    en_static_define_state_off                      : INT;   // Definierter State für OFF-Zustand
    en_static_define_sub_state_off                  : INT;   // Definierter Substate für OFF-Zustand
    en_static_define_lockdown                       : INT;   // State für Lockdown-Bedingungen
    en_static_define_substate_check_new_state       : INT;   // Substate zur Prüfung eines neuen State
    en_static_define_engine_release_from_substate   : INT;   // Substate, wenn Engine in Release-ON gehen soll
	en_static_define_engine_release_off_substate    : INT;   // Substate, wenn Engine in Release-OFF gehen soll
END_VAR

VAR_OUTPUT
    iAvaiable                                       : INT;   // Verfügbarkeitskennzahl der Engine/Gruppe
    en_available                                    : INT;   // Haupt-State der Verfügbarkeit
    en_available_substate                           : INT;   // Substate der Verfügbarkeit

    iAcknowledge                                    : INT;   // Integer-Wert zur Acknowledge-Verarbeitung
    rAcknowledge                                    : REAL;  // Realwert für Acknowledge-Parameter
    en_acknowledge                                  : INT;   // State für Acknowledge-Vorgang
    en_acknowledge_substate                         : INT;   // Substate des Acknowledge-Vorgangs

    en_demand                                       : INT;   // Haupt-State für Demand-/Anforderung
    en_demand_substate                              : INT;   // Substate für Demand-/Anforderung
    
    ITF_MANAGER                                     : ITF_MANAGER; // Manager-Interface für Gruppen-/Engine-Steuerung
END_VAR

VAR
    aydiSyncG                                       : ARRAY[1..GVL_CONSTANT.MAX_GROUPS] OF DINT := [GVL_CONSTANT.MAX_GROUPS(1)];
                                                        // Array zur Synchronisationsverwaltung der Gruppen

    groups                                          : ARRAY[1..GVL_CONSTANT.MAX_GROUPS] OF ARRAY[0..40] OF ITF_GROUPBASE;
                                                        // Struktur aller Gruppen und ihrer Members

    groups_en_available                             : ARRAY[1..GVL_CONSTANT.MAX_GROUPS] OF INT; // Verfügbarkeits-State je Gruppe
    groups_en_available_old                         : ARRAY[1..GVL_CONSTANT.MAX_GROUPS] OF INT; // Vorheriger Verfügbarkeits-State
    groups_en_available_substate                    : ARRAY[1..GVL_CONSTANT.MAX_GROUPS] OF INT; // Verfügbarkeits-Substate je Gruppe
    groups_en_available_substate_old                : ARRAY[1..GVL_CONSTANT.MAX_GROUPS] OF INT; // Alter Substate

    groups_engine_avaiable                          : ARRAY[1..GVL_CONSTANT.MAX_GROUPS] OF INT; // Engine-Verfügbarkeitsstate je Gruppe

    groups_en_acknowledge                           : ARRAY[1..GVL_CONSTANT.MAX_GROUPS] OF INT; // Acknowledge-State je Gruppe
    groups_en_acknowledge_old                       : ARRAY[1..GVL_CONSTANT.MAX_GROUPS] OF INT; // Alter Acknowledge-State
    groups_en_acknowledge_substate                  : ARRAY[1..GVL_CONSTANT.MAX_GROUPS] OF INT; // Acknowledge-Substate je Gruppe
    groups_en_acknowledge_substate_old              : ARRAY[1..GVL_CONSTANT.MAX_GROUPS] OF INT; // Alter Acknowledge-Substate

    groups_engine_acknowledge                       : ARRAY[1..GVL_CONSTANT.MAX_GROUPS] OF INT; // Engine-Acknowledge-State je Gruppe

    groups_en_release                               : ARRAY[1..GVL_CONSTANT.MAX_GROUPS] OF INT; // Release-State je Gruppe

    AY_GROUPS_AyPosMaxCT                            : ARRAY[1..GVL_CONSTANT.MAX_GROUPS] OF DINT; // Max-CT-Werte der Gruppen
    AY_GROUPS_xReleaseCircuit                       : ARRAY[1..GVL_CONSTANT.MAX_GROUPS] OF BOOL; // Release-Freigabe je Circuit

    TEMP_ITF_GROUPBASE                              : ITF_GROUPBASE; // Temp-Objekt für Gruppenoperationen
    TEMP_ITF_CIRCUIT                                : ITF_CIRCUIT;    // Temp-Circuit-Objekt
    TEMP_ITF_HYDRA                                  : ITF_HYDRA;      // Temp-Hydra-Objekt
    TEMP_ITF_HYDRA_MAX_CT                           : ITF_HYDRA;      // Temp-Hydra Objekt für max CT-Ermittlung

    diTempMemberCount                                : DINT;  // Temporäre Anzahl an Gruppenmitgliedern
    diFor1                                           : DINT;  // Schleifenzähler 1
    diFor2                                           : DINT;  // Schleifenzähler 2
    diFor3                                           : DINT;  // Schleifenzähler 3
    diNextCircuitToRun                               : DINT;  // Nächster Circuit, der gestartet werden soll
    diNextEngineToRun                                : DINT;  // Nächste Engine, die starten soll
    diNextCircuitToOff                               : DINT;  // Nächster Circuit zum Ausschalten
    diNextEngineToOff                                : DINT;  // Nächste Engine zum Ausschalten

    xTrigOn                                          : BOOL;  // Trigger für Start-/ON-Übergang
    xTrigOff                                         : BOOL;  // Trigger für Stop-/OFF-Übergang
    iTrigOffCount                                    : INT;   // Zähler für OFF-Triggerpflege
    iTrigOffMax                                      : INT;   // Maximal zulässige OFF-Triggerzeit

    enCheckOld                                       : INT;   // Alter Check-State
    enReleaseOld                                     : INT;   // Alter Release-State

    uiCountGroupLockDown                             : UINT;  // Anzahl Gruppen im Lockdown
    uiCountEngineLockDown                            : UINT;  // Anzahl Engines im Lockdown
    uiCountEngineAcknowledge                         : UINT;  // Anzahl Engines, die Acknowledge benötigen
    uiCountGroupLockDownOld                          : UINT;  // Vorherige Lockdown-Gruppenzahl
    uiCountEngineAcknowledgeOld                      : UINT;  // Vorherige Anzahl Acknowledge-Engines
    uiCountEngineLockDownOld                         : UINT;  // Vorherige Lockdown-Enginezahl

    iReleaseOld                                      : INT;   // Alter Releasewert
    iAcknowledgeOld                                  : INT;   // Alter Acknowledgewert

    xReleaseStopp                                    : BOOL;  // Stopp-Bedingung für Release
    TP_ReleaseLock                                   : Standard.TP;   // Timerbaustein für Release-Lock
    xResettReleaseLock_VIS                           : BOOL;  // Reset über VIS zum ReleaseLock

    lock_if_released_in_other_circuit                : BOOL;  // Lock, wenn Release in anderem Circuit aktiv ist

    // Parameter
    fbConfigFile                                     : CtaSysConfig.fbConfigFile; // Konfigurationsdatei-Handler
    scParameter                                      : scParameter;               // Parametrierobjekt
END_VAR

actParameter();

(* ITF *)
ITF_MANAGER := THIS^;

(* CHECK *)
CHECK();

(* AVAIABLE *)
AVAIABLE(); 

(* LOCKDOWN *)
LOCKDOWN();

(* ACKNOWLEDGE *)
ACKNOWLEDGE();

(* MANAGEMENT *)
MANAGEMENT();

(* RELEASE *)
RELEASE();

(* CHECK CHANGE *)
CHECK_RELEASE_CHANGE();

(* UPDATE *)
UPDATE_AT_THE_END();

ACTION CHECK:
(* Set Check State *)
FOR diFor1 := LOWER_BOUND(groups,1) TO UPPER_BOUND(groups,1) DO
	FOR diFor2 := LOWER_BOUND(groups[diFor1],1) TO UPPER_BOUND(groups[diFor1],1) DO
		IF __QUERYINTERFACE(groups[diFor1][diFor2],TEMP_ITF_GROUPBASE) THEN
			TEMP_ITF_GROUPBASE.set_check			(en_check);
			TEMP_ITF_GROUPBASE.set_check_substate	(en_check_substate);
		END_IF;
	END_FOR;
END_FOR;
END_ACTION

METHOD GET_NEXT_ENGINE_TO_RUN 
VAR_INPUT
	enTYPE_OF_ENGINE_MANAGEMENT	:	TYPE_OF_ENGINE_MANAGEMENT;
END_VAR
VAR_OUTPUT
	diNextCircuitToRunOut  		: DINT;
	diNextEngineToRunOut		: DINT;	
END_VAR
VAR 
	_diNextCircuitToRun  		: DINT;
	_diEngineLowestRunTime		: DINT;
	_xAvaiable					: BOOL;
	_xRelease					: BOOL;
	_rRelease					: REAL;
	_xAcknowledge				: BOOL;
	_rAcknowledge				: REAL;
	_xLockDown					: BOOL;
	_udiRunTime		    		: UDINT;
	_udiRunTimeTillOn   		: UDINT;
	_udiMinRunTime				: UDINT;
	_uiLowestWorkloadCircuit	: UINT;
END_VAR
(* Set Min Run Time To Max *)
_udiMinRunTime := 16#FFFFFFFF;
(* Set Lowest Workload Circuit to MAX *)
_uiLowestWorkloadCircuit := 16#FFFF;
(* Set Circuit to 0 *)
_diNextCircuitToRun := 0;
diNextCircuitToRunOut := 0;
(* Set Engine to 0  *)
_diEngineLowestRunTime := 0;
diNextEngineToRunOut := 0;

IF enTYPE_OF_ENGINE_MANAGEMENT = TYPE_OF_ENGINE_MANAGEMENT.RUN_1BY1 THEN
	FOR diFor1 := UPPER_BOUND(groups,1) TO LOWER_BOUND(groups,1) BY -1 DO 
		(* If No Error avaiable to release*)
		IF groups_en_available[diFor1] = en_release  OR groups_en_acknowledge[diFor1] = en_release THEN		
			IF __QUERYINTERFACE(groups[diFor1][LOWER_BOUND(groups[diFor1],1)],TEMP_ITF_CIRCUIT) THEN
				IF TEMP_ITF_CIRCUIT.GET_ANZ_RELEASE > 0 AND TEMP_ITF_CIRCUIT.GET_ANZ_AVAIABLE > 0 THEN
					(* iterate Engine and Check if Avaiable and get the Minits *)
					FOR diFor2 := TEMP_ITF_CIRCUIT.UPPERBOUND TO TEMP_ITF_CIRCUIT.LOWERBOUND BY -1 DO
						TEMP_ITF_CIRCUIT.GET_ENGINE_STATE(	usiNr 			:= TO_USINT(diFor2),
															xAvaiable 		=> _xAvaiable,
															xRelease		=> _xRelease,
															rRelease		=> _rRelease,
															xAcknowledge 	=> _xAcknowledge,
															rAcknowledge 	=> _rAcknowledge,
															xLockDown 		=> _xLockDown,
															udiRunTime 		=> _udiRunTime,
															udiRunTimeTillOn=> _udiRunTimeTillOn);
						(* Get time if Avaiable *)
						IF _xAvaiable AND NOT _xRelease AND NOT _xLockDown THEN
							IF _udiRunTime <= _udiMinRunTime THEN
								_udiMinRunTime 			:= _udiRunTime;
								_diNextCircuitToRun 	:= diFor1;
								_diEngineLowestRunTime  := diFor2;
							END_IF;			
						END_IF;						
					END_FOR;
				END_IF;
			END_IF;
		END_IF;
	END_FOR;
	(* Get new Ccuit if not possible to add ad running circuti *)
	IF _diNextCircuitToRun = 0 AND _diEngineLowestRunTime = 0  THEN
		FOR diFor1 := UPPER_BOUND(groups,1) TO LOWER_BOUND(groups,1) BY -1 DO
			(* If No Error avaiable to release*)
			IF groups_en_available[diFor1] = en_release  OR groups_en_acknowledge[diFor1] = en_release THEN	
				IF __QUERYINTERFACE(groups[diFor1][LOWER_BOUND(groups[diFor1],1)],TEMP_ITF_CIRCUIT) THEN
					IF TEMP_ITF_CIRCUIT.GET_ANZ_AVAIABLE > 0 THEN
						(* iterate Engine and Check if Avaiable and get the Minits *)
						FOR diFor2 := TEMP_ITF_CIRCUIT.UPPERBOUND TO TEMP_ITF_CIRCUIT.LOWERBOUND BY -1 DO
							TEMP_ITF_CIRCUIT.GET_ENGINE_STATE(	usiNr 			:= TO_USINT(diFor2),
																xAvaiable 		=> _xAvaiable,
																xRelease		=> _xRelease,
																rRelease		=> _rRelease,
																xAcknowledge 	=> _xAcknowledge,
																rAcknowledge 	=> _rAcknowledge,
																xLockDown 		=> _xLockDown,
																udiRunTime 		=> _udiRunTime,
																udiRunTimeTillOn=> _udiRunTimeTillOn);
							(* Get time if Avaiable *)
							IF _xAvaiable AND NOT _xRelease AND NOT _xLockDown THEN
								IF _udiRunTime <= _udiMinRunTime THEN
									_udiMinRunTime 			:= _udiRunTime;
									_diNextCircuitToRun 	:= diFor1;
									_diEngineLowestRunTime  := diFor2;
								END_IF;			
							END_IF;						
						END_FOR;
					END_IF;
				END_IF;
			END_IF;
		END_FOR;		
	END_IF
(* EQUAL *)
ELSIF enTYPE_OF_ENGINE_MANAGEMENT = TYPE_OF_ENGINE_MANAGEMENT.RUN_EQUAL THEN
	FOR diFor1 := UPPER_BOUND(groups,1) TO LOWER_BOUND(groups,1) BY -1 DO 
		(* If No Error avaiable to release*)
		IF groups_en_available[diFor1] = en_release  OR groups_en_acknowledge[diFor1] = en_release THEN	
			IF __QUERYINTERFACE(groups[diFor1][LOWER_BOUND(groups[diFor1],1)],TEMP_ITF_CIRCUIT) THEN
				IF TEMP_ITF_CIRCUIT.GET_ANZ_RELEASE <= _uiLowestWorkloadCircuit AND TEMP_ITF_CIRCUIT.GET_ANZ_AVAIABLE > 0 THEN
					_uiLowestWorkloadCircuit := TEMP_ITF_CIRCUIT.GET_ANZ_RELEASE; 
					(* iterate Engine and Check if Avaiable and get the Minits *)
					FOR diFor2 := TEMP_ITF_CIRCUIT.UPPERBOUND TO TEMP_ITF_CIRCUIT.LOWERBOUND BY -1 DO
						TEMP_ITF_CIRCUIT.GET_ENGINE_STATE(	usiNr 			:= TO_USINT(diFor2),
															xAvaiable 		=> _xAvaiable,
															xRelease		=> _xRelease,
															rRelease		=> _rRelease,
															xAcknowledge 	=> _xAcknowledge,
															rAcknowledge 	=> _rAcknowledge,
															xLockDown 		=> _xLockDown,
															udiRunTime 		=> _udiRunTime,
															udiRunTimeTillOn=> _udiRunTimeTillOn);
						(* Get time if Avaiable *)
						IF _xAvaiable AND NOT _xRelease AND NOT _xLockDown THEN
							IF _udiRunTime <= _udiMinRunTime THEN
								_udiMinRunTime 			:= _udiRunTime;
								_diNextCircuitToRun 	:= diFor1;
								_diEngineLowestRunTime  := diFor2;
							END_IF;			
						END_IF;						
					END_FOR;
				END_IF;
			END_IF;
		END_IF;
	END_FOR;
END_IF;
diNextCircuitToRunOut 	:= _diNextCircuitToRun;
diNextEngineToRunOut	:= _diEngineLowestRunTime;
END_METHOD

METHOD GET_NEXT_ENGINE_TO_OFF 
VAR_INPUT
	enTYPE_OF_ENGINE_MANAGEMENT	:	TYPE_OF_ENGINE_MANAGEMENT;
END_VAR
VAR_OUTPUT
	diNextCircuitToOffOut  		: DINT;
	diNextEngineToOffOut		: DINT;	
END_VAR
VAR 
	_diNextCircuitToOff  		: DINT;
	_diEngineHighestRunTime		: DINT;
	_xAvaiable					: BOOL;
	_xRelease					: BOOL;
	_rRelease					: REAL;
	_xAcknowledge				: BOOL;
	_rAcknowledge				: REAL;
	_xLockDown					: BOOL;
	_udiRunTime		    		: UDINT;
	_udiRunTimeTillOn   		: UDINT;
	_udiMaxRunTimeTillOn		: UDINT;
	_uiHighestWorkloadCircuit	: UINT;
	_uiLowestWorkloadCircuit	: UINT;
END_VAR
(* Set Highest Workload Circuit to Min *)
_uiHighestWorkloadCircuit := 16#0000;
(* Set Lowest Workload Circuit to MAX *)
_uiLowestWorkloadCircuit := 16#FFFF;
(* Set Max Run Time To Min *)
_udiMaxRunTimeTillOn := 16#0000;
(* Set Circuit to 0 *)
_diNextCircuitToOff := 0;
diNextCircuitToOffOut := 0;
(* Set Engine to 0  *)
_diEngineHighestRunTime := 0;
diNextEngineToOffOut := 0;
(* 1By1 *)
IF enTYPE_OF_ENGINE_MANAGEMENT = TYPE_OF_ENGINE_MANAGEMENT.RUN_1BY1 THEN
	FOR diFor1 := UPPER_BOUND(groups,1) TO LOWER_BOUND(groups,1) BY -1 DO 
		(* If No Error avaiable to release*)
		IF groups_en_available[diFor1] = en_release  OR groups_en_acknowledge[diFor1] = en_release THEN	
			IF __QUERYINTERFACE(groups[diFor1][LOWER_BOUND(groups[diFor1],1)],TEMP_ITF_CIRCUIT) THEN
				IF TEMP_ITF_CIRCUIT.GET_ANZ_RELEASE > 0 THEN
					IF TEMP_ITF_CIRCUIT.GET_ANZ_RELEASE <= _uiLowestWorkloadCircuit THEN
						IF TEMP_ITF_CIRCUIT.GET_ANZ_RELEASE < _uiLowestWorkloadCircuit THEN
							_uiLowestWorkloadCircuit := TEMP_ITF_CIRCUIT.GET_ANZ_RELEASE; 
							(* Set Max Run Time To Min *)
							_udiMaxRunTimeTillOn := 16#0000;
						END_IF;

						(* iterate Engine and Check if Avaiable and get the Minits *)
						FOR diFor2 := TEMP_ITF_CIRCUIT.UPPERBOUND TO TEMP_ITF_CIRCUIT.LOWERBOUND BY -1 DO
							TEMP_ITF_CIRCUIT.GET_ENGINE_STATE(	usiNr 			:= TO_USINT(diFor2),
																xAvaiable 		=> _xAvaiable,
																xRelease		=> _xRelease,
																rRelease		=> _rRelease,
																xAcknowledge 	=> _xAcknowledge,
																rAcknowledge 	=> _rAcknowledge,
																xLockDown 		=> _xLockDown,
																udiRunTime 		=> _udiRunTime,
																udiRunTimeTillOn=> _udiRunTimeTillOn);
							(* Get time if Running *)
							IF _xRelease THEN
								IF _udiRunTimeTillOn >= _udiMaxRunTimeTillOn THEN
									_udiMaxRunTimeTillOn 	:= _udiRunTimeTillOn;
									_diNextCircuitToOff 	:= diFor1;
									_diEngineHighestRunTime := diFor2;
								END_IF;			
							END_IF;						
						END_FOR;
					END_IF;
				END_IF;
			END_IF;
		END_IF;
	END_FOR;
(* EQUAL *)
ELSIF enTYPE_OF_ENGINE_MANAGEMENT = TYPE_OF_ENGINE_MANAGEMENT.RUN_EQUAL THEN
	FOR diFor1 := UPPER_BOUND(groups,1) TO LOWER_BOUND(groups,1) BY -1 DO 
		(* If No Error avaiable to release*)
		IF groups_en_available[diFor1] = en_release OR groups_en_acknowledge[diFor1] = en_release THEN	
			IF __QUERYINTERFACE(groups[diFor1][LOWER_BOUND(groups[diFor1],1)],TEMP_ITF_CIRCUIT) THEN
				IF TEMP_ITF_CIRCUIT.GET_ANZ_RELEASE >= _uiHighestWorkloadCircuit THEN
					IF TEMP_ITF_CIRCUIT.GET_ANZ_RELEASE > _uiHighestWorkloadCircuit THEN
						_uiHighestWorkloadCircuit := TEMP_ITF_CIRCUIT.GET_ANZ_RELEASE; 
						(* Set Max Run Time To Min *)
						_udiMaxRunTimeTillOn := 16#0000;				
					END_IF;
					(* iterate Engine and Check if Avaiable and get the time *)
					FOR diFor2 := TEMP_ITF_CIRCUIT.UPPERBOUND TO TEMP_ITF_CIRCUIT.LOWERBOUND BY -1 DO
						TEMP_ITF_CIRCUIT.GET_ENGINE_STATE(	usiNr 			:= TO_USINT(diFor2),
															xAvaiable 		=> _xAvaiable,
															xRelease		=> _xRelease,
															rRelease		=> _rRelease,
															xAcknowledge 	=> _xAcknowledge,
															rAcknowledge 	=> _rAcknowledge,
															xLockDown 		=> _xLockDown,
															udiRunTime 		=> _udiRunTime,
															udiRunTimeTillOn=> _udiRunTimeTillOn);
						(* Get time if Running *)
						IF _xRelease THEN
							IF _udiRunTimeTillOn >= _udiMaxRunTimeTillOn THEN
								_udiMaxRunTimeTillOn 	:= _udiRunTimeTillOn;
								_diNextCircuitToOff 	:= diFor1;
								_diEngineHighestRunTime := diFor2;
							END_IF;			
						END_IF;						
					END_FOR;
				END_IF;
			END_IF;
		END_IF;
	END_FOR;
END_IF;
diNextCircuitToOffOut 	:= _diNextCircuitToOff;
diNextEngineToOffOut	:= _diEngineHighestRunTime;
END_METHOD

ACTION MANAGEMENT:
(* ------------------------------------------------------------- *)
(* Engine Trigger Logic: TRIG ON / TRIG OFF and Release Handling   *)
(* ------------------------------------------------------------- *)

(* Wait until no TRIG ON is active, then determine next engine to run *)
IF NOT xTrigOn THEN
    GET_NEXT_ENGINE_TO_RUN(
        enTYPE_OF_ENGINE_MANAGEMENT := scParameter.fbiTypeOfEngineManagement.proValue,
        diNextCircuitToRunOut => diNextCircuitToRun,
        diNextEngineToRunOut  => diNextEngineToRun
    );
END_IF;

(* Wait until no TRIG OFF is active, then determine next engine to stop *)
IF NOT xTrigOff THEN
    GET_NEXT_ENGINE_TO_OFF(
        enTYPE_OF_ENGINE_MANAGEMENT := scParameter.fbiTypeOfEngineManagement.proValue,
        diNextCircuitToOffOut => diNextCircuitToOff,
        diNextEngineToOffOut  => diNextEngineToOff
    );
END_IF;

(* Check if engine is available and TRIG ON conditions are met *)
IF diNextCircuitToRun > 0 AND diNextEngineToRun > 0 THEN
    IF xRelease AND iRelease > 0 AND NOT xReleaseStopp THEN

        (* Handle group lockdown events *)
        IF uiCountGroupLockDown > uiCountGroupLockDownOld AND en_acknowledge <> en_static_define_lockdown THEN
            xTrigOn := TRUE;
            TP_ReleaseLock(IN := FALSE);

        (* Handle engine lockdown events *)
        ELSIF uiCountEngineLockDown > uiCountEngineLockDownOld AND en_acknowledge <> en_static_define_lockdown THEN
            xTrigOn := TRUE;
            TP_ReleaseLock(IN := FALSE);

        (* Handle engine turning off unexpectedly *)
        ELSIF uiCountEngineAcknowledge < uiCountEngineAcknowledgeOld AND iRelease > TO_INT(uiCountEngineAcknowledge) AND en_acknowledge <> en_static_define_lockdown THEN
            xTrigOn := TRUE;
            TP_ReleaseLock(IN := FALSE);

        (* Normal case: Add engine if release request exceeds acknowledge and no lock active *)
        ELSIF iRelease > iAcknowledge AND NOT TP_ReleaseLock.Q AND NOT xTrigOn THEN
            TP_ReleaseLock(IN := FALSE); (* Reset pulse before trigger *)
            xTrigOn := TRUE;
        END_IF;

    ELSE
        xTrigOn := FALSE; (* Release not active → no TRIG ON *)
    END_IF;
END_IF;

(* Manage normal release lock timer with minimum of 60s *)
IF NOT xResettReleaseLock_VIS AND xRelease THEN
    IF scParameter.fbtZuschaltSperrzeit.proValue > T#60S THEN
        TP_ReleaseLock(PT := scParameter.fbtZuschaltSperrzeit.proValue);
    ELSE
        TP_ReleaseLock(PT := T#60S);
    END_IF;
ELSE
    TP_ReleaseLock(IN := FALSE, PT := T#0MS);
    xResettReleaseLock_VIS := FALSE;
END_IF;

(* Check if engine is available and TRIG OFF conditions are met *)
IF diNextCircuitToOff > 0 AND diNextEngineToOff > 0 THEN
    IF xRelease THEN

        (* Reset case: Release equals acknowledge → reset counters *)
        IF iRelease = iAcknowledge THEN
            iTrigOffMax := 0;
            iTrigOffCount := 0;
            IF xTrigOn THEN (* Prevent endless engine running *)
                xTrigOn := FALSE;
                xTrigOff := TRUE;
                diNextCircuitToOff := diNextCircuitToRun;
                diNextEngineToOff  := diNextEngineToRun;
            END_IF

        (* Normal reduction: Release < acknowledge → trigger engine off *)
        ELSIF iRelease < iAcknowledge THEN
            IF iRelease < iReleaseOld OR iAcknowledge > iAcknowledgeOld THEN
                iTrigOffMax := MIN(iAcknowledge, iTrigOffMax + iReleaseOld - iRelease);
            END_IF
            IF iTrigOffCount < iTrigOffMax THEN
                iTrigOffCount := iTrigOffCount + 1;
                xTrigOff := TRUE;
            END_IF;
        END_IF;

    ELSE
        xTrigOff := FALSE; (* Release inactive → no TRIG OFF *)
    END_IF;
END_IF;

(* Set Release array and trigger engines accordingly *)
FOR diFor1 := LOWER_BOUND(groups,1) TO UPPER_BOUND(groups,1) DO
    IF __QUERYINTERFACE(groups[diFor1][LOWER_BOUND(groups[diFor1],1)], TEMP_ITF_CIRCUIT) THEN
        IF groups_en_acknowledge[diFor1] <> en_static_define_lockdown THEN
            IF TEMP_ITF_CIRCUIT.IS_RELEVANT_TO_RELEASE THEN

                (* Stop engine if it is next to be turned off *)
                IF diFor1 = diNextCircuitToOff AND xTrigOff THEN
                    TEMP_ITF_CIRCUIT.RELEASE_ENGINE(TO_USINT(diNextEngineToOff), FALSE);
                    xTrigOff := FALSE;
                    xTrigOn := FALSE;
                END_IF;

                (* Release engine if it is next to run and TRIG ON is active *)
                IF (groups_en_available[diFor1] = en_release OR groups_en_available[diFor1] = en_release_next OR groups_en_acknowledge[diFor1] = en_release) AND diFor1 = diNextCircuitToRun AND xTrigOn AND iRelease > 0 THEN
                    groups_en_release[diFor1] := en_release;
                    IF groups_en_acknowledge_substate[diFor1] >= en_static_define_engine_release_from_substate AND groups_en_acknowledge_substate[diFor1] <= en_static_define_engine_release_off_substate THEN
                        IF TEMP_ITF_CIRCUIT.IS_RELEVANT_TO_RELEASE AND AY_GROUPS_xReleaseCircuit[diFor1] THEN
							TEMP_ITF_CIRCUIT.RELEASE_ENGINE(TO_USINT(diNextEngineToRun), TRUE);
						END_IF;
                        xTrigOn := FALSE;
                        TP_ReleaseLock(IN := TRUE);
                    ELSE
                        TEMP_ITF_CIRCUIT.ALL_OFF();
                    END_IF;
                ELSIF groups_en_acknowledge[diFor1] = en_static_define_lockdown OR TEMP_ITF_CIRCUIT.GET_ANZ_RELEASE = 0 OR iRelease = 0 OR groups_en_acknowledge_substate[diFor1] < en_static_define_engine_release_from_substate OR groups_en_acknowledge_substate[diFor1] > en_static_define_engine_release_off_substate THEN
                    TEMP_ITF_CIRCUIT.ALL_OFF();
                    groups_en_release[diFor1] := en_static_define_state_off;
                END_IF;

            ELSE
                TEMP_ITF_CIRCUIT.ALL_OFF();
                groups_en_release[diFor1] := en_release;
            END_IF;
        ELSE
            TEMP_ITF_CIRCUIT.ALL_OFF();
            groups_en_release[diFor1] := en_static_define_state_off;
        END_IF;
    ELSE
        groups_en_release[diFor1] := en_static_define_state_off;
    END_IF;
END_FOR;

(* Apply HZ scale to relevant circuits *)
FOR diFor1 := LOWER_BOUND(groups,1) TO UPPER_BOUND(groups,1) DO
    IF __QUERYINTERFACE(groups[diFor1][LOWER_BOUND(groups[diFor1],1)], TEMP_ITF_CIRCUIT) THEN
        IF TEMP_ITF_CIRCUIT.IS_RELEVANT_TO_RELEASE THEN
            TEMP_ITF_CIRCUIT.SET_HZ_SCALE(scHzRelease);
        END_IF;
    END_IF;
END_FOR;

(* Set cyclic speed proportionally if acknowledge has not changed *)
IF iAcknowledge = iAcknowledgeOld THEN
    FOR diFor1 := LOWER_BOUND(groups,1) TO UPPER_BOUND(groups,1) DO
        IF __QUERYINTERFACE(groups[diFor1][LOWER_BOUND(groups[diFor1],1)], TEMP_ITF_CIRCUIT) THEN
            IF TEMP_ITF_CIRCUIT.IS_RELEVANT_TO_RELEASE THEN
                FOR diFor2 := TEMP_ITF_CIRCUIT.LOWERBOUND TO TEMP_ITF_CIRCUIT.UPPERBOUND DO
                    TEMP_ITF_CIRCUIT.prorRelease := rRelease;
                END_FOR;
            END_IF;
        END_IF;
    END_FOR;
END_IF;
END_ACTION

ACTION CHECK_RELEASE_CHANGE:
(* Not Avaiable if Changed *)
IF en_check <> enCheckOld THEN
	en_available := en_static_define_substate_check_new_state;
END_IF;
END_ACTION

ACTION UPDATE_AT_THE_END:
iAcknowledgeOld := iAcknowledge;
enReleaseOld 	:= en_release;
enCheckOld	 	:= en_check;
iReleaseOld		:= iRelease;
END_ACTION

ACTION ACKNOWLEDGE:
(* ------------------------------------------------------------- *)
(* Reset Phase: Initialize group acknowledge status variables      *)
(* ------------------------------------------------------------- *)
FOR diFor1 := LOWER_BOUND(groups,1) TO UPPER_BOUND(groups,1) DO
    IF __QUERYINTERFACE(groups[diFor1][0], TEMP_ITF_CIRCUIT) THEN
        (* Set initial acknowledge state to release for circuits *)
        groups_en_acknowledge[diFor1] := en_release;
        groups_en_acknowledge_substate[diFor1] := en_release_substate;
    ELSE
        (* Set initial acknowledge state to Lockdown if no circuit *)
        groups_en_acknowledge[diFor1] := en_static_define_lockdown;
        groups_en_acknowledge_substate[diFor1] := en_static_define_sub_state_off;
    END_IF;
END_FOR;

(* ------------------------------------------------------------- *)
(* Determine actual acknowledge status of each group               *)
(* ------------------------------------------------------------- *)
FOR diFor1 := LOWER_BOUND(groups,1) TO UPPER_BOUND(groups,1) DO
    (* Iterate over all members of the group *)
    FOR diFor2 := LOWER_BOUND(groups[diFor1],1) TO UPPER_BOUND(groups[diFor1],1) DO
        IF __QUERYINTERFACE(groups[diFor1][diFor2], groups[diFor1][diFor2]) THEN
            (* Only consider relevant objects for release and acknowledge *)
            IF NOT groups[diFor1][diFor2].IS_NOT_RELEVANT_TO_RELEASE AND NOT groups[diFor1][diFor2].IS_NOT_RELEVANT_TO_ACKNOWLEDGE THEN
                (* Update group acknowledge status based on member *)
                IF groups[diFor1][diFor2].acknowledge <> en_release THEN
                    IF groups[diFor1][diFor2].acknowledge = en_static_define_lockdown THEN
                        (* If this group was about to run, cancel TRIG ON *)
                        IF diNextCircuitToRun = diFor1 AND xTrigOn THEN
                            xTrigOn := FALSE;
                        END_IF;
                        groups_en_acknowledge[diFor1] := en_static_define_lockdown; (* Lockdown for group *)
                    ELSE
						IF groups_en_acknowledge[diFor1] <> en_static_define_lockdown THEN
                        	groups_en_acknowledge[diFor1] := groups[diFor1][diFor2].acknowledge;
						END_IF;
                    END_IF;
                END_IF;

                (* Update substate if it differs from release substate *)
                IF groups[diFor1][diFor2].acknowledge_substate <> en_release_substate THEN
                    groups_en_acknowledge_substate[diFor1] := groups[diFor1][diFor2].acknowledge_substate;
                END_IF;
            END_IF;
        END_IF;
    END_FOR;

    (* Count acknowledged engines per group if circuit interface is valid *)
    IF __QUERYINTERFACE(groups[diFor1][LOWER_BOUND(groups[diFor1],1)], TEMP_ITF_CIRCUIT) THEN
        groups_engine_acknowledge[diFor1] := TO_INT(TEMP_ITF_CIRCUIT.GET_ANZ_ACKNOWLEDGE);
    ELSE
        groups_engine_acknowledge[diFor1] := 0;
    END_IF;
END_FOR;

(* ------------------------------------------------------------- *)
(* Set acknowledge status for manager based on group status       *)
(* ------------------------------------------------------------- *)
en_acknowledge := 0;
FOR diFor1 := LOWER_BOUND(groups,1) TO UPPER_BOUND(groups,1) DO
    (* If any group is in lockdown, manager is in lockdown *)
    IF groups_en_acknowledge[diFor1] = en_static_define_lockdown THEN
        en_acknowledge := en_static_define_lockdown;
    END_IF;
END_FOR;

FOR diFor1 := LOWER_BOUND(groups,1) TO UPPER_BOUND(groups,1) DO
    (* If any group is in release and substate matches, update manager acknowledge *)
    IF groups_en_acknowledge[diFor1] = en_release OR ( groups_en_acknowledge[diFor1] <> en_static_define_lockdown AND groups_en_release[diFor1] = en_release ) THEN
		en_acknowledge := groups_en_acknowledge[diFor1];
        IF groups_en_acknowledge_substate[diFor1] = en_release_substate  THEN
            en_acknowledge_substate := en_release_substate;
        END_IF;		
    END_IF;
END_FOR;

(* Update engine acknowledge counters *)
iAcknowledge := 0;
uiCountEngineAcknowledgeOld := uiCountEngineAcknowledge;
FOR diFor1 := LOWER_BOUND(groups,1) TO UPPER_BOUND(groups,1) DO
    iAcknowledge := iAcknowledge + groups_engine_acknowledge[diFor1];
END_FOR;
uiCountEngineAcknowledge := TO_UINT(iAcknowledge);
END_ACTION

ACTION RELEASE:
(* Set Release for each group and its components *)
FOR diFor1 := LOWER_BOUND(groups,1) TO UPPER_BOUND(groups,1) DO

    (* Check if group is in release state and not in lockdown *)
    IF groups_en_release[diFor1] = en_release AND groups_en_acknowledge[diFor1] <> en_static_define_lockdown THEN
        (* Initially set group as ready for release *)
        AY_GROUPS_xReleaseCircuit[diFor1] := TRUE;

        (* Check each member in the group to verify readiness for release *)
        FOR diFor2 := LOWER_BOUND(groups[diFor1],1)+1 TO UPPER_BOUND(groups[diFor1],1) DO
            IF __QUERYINTERFACE(groups[diFor1][diFor2], TEMP_ITF_HYDRA) THEN
                IF NOT groups[diFor1][diFor2].IS_NOT_RELEVANT_TO_RELEASE AND NOT groups[diFor1][diFor2].IS_NOT_RELEVANT_TO_ACKNOWLEDGE THEN
                    IF groups[diFor1][diFor2].acknowledge <> en_release OR groups[diFor1][diFor2].acknowledge_substate <> en_static_define_engine_release_from_substate THEN
                        (* Member not ready, set group as not ready *)
                        AY_GROUPS_xReleaseCircuit[diFor1] := FALSE;
                    END_IF;
                END_IF;
            END_IF;
        END_FOR;

        (* Apply release settings to each relevant member of the group *)
        FOR diFor2 := LOWER_BOUND(groups[diFor1],1)+1 TO UPPER_BOUND(groups[diFor1],1) DO
            IF __QUERYINTERFACE(groups[diFor1][diFor2], groups[diFor1][diFor2]) THEN
                IF NOT groups[diFor1][diFor2].IS_NOT_RELEVANT_TO_RELEASE THEN
                    IF __QUERYINTERFACE(groups[diFor1][diFor2], TEMP_ITF_HYDRA) THEN
                        TEMP_ITF_HYDRA.set_release(en_release);
                        TEMP_ITF_HYDRA.set_release_substate(en_release_substate);
                        TEMP_ITF_HYDRA.set_release_next(en_release_next);
                    END_IF;
                ELSE
                    (* Member not relevant → set off *)
                    IF __QUERYINTERFACE(groups[diFor1][diFor2], TEMP_ITF_HYDRA) THEN
                        TEMP_ITF_HYDRA.set_release(en_static_define_state_off);
                        TEMP_ITF_HYDRA.set_release_substate(en_static_define_sub_state_off);
                        TEMP_ITF_HYDRA.set_release_next(en_release_next);
                    END_IF;
                END_IF;
            END_IF;
        END_FOR;

        (* Release settings for group leader *)
        IF groups[diFor1][LOWER_BOUND(groups[diFor1],1)] <> 0 THEN
            IF __QUERYINTERFACE(groups[diFor1][LOWER_BOUND(groups[diFor1],1)], TEMP_ITF_CIRCUIT) THEN
				TEMP_ITF_CIRCUIT.set_release(en_release);
				TEMP_ITF_CIRCUIT.set_release_substate(en_release_substate);
				TEMP_ITF_CIRCUIT.set_release_next(en_release_next);
			ELSE
				(* Leader not relevant → set off *)
				TEMP_ITF_CIRCUIT.set_release(en_release);
				TEMP_ITF_CIRCUIT.set_release_substate(en_release_substate);
				TEMP_ITF_CIRCUIT.set_release_next(en_release_next);
			END_IF;
        END_IF;

    ELSE
        (* Group not in release → mark as not ready *)
        AY_GROUPS_xReleaseCircuit[diFor1] := FALSE;

        (* Turn off all members of the group *)
        FOR diFor2 := LOWER_BOUND(groups[diFor1],1) TO UPPER_BOUND(groups[diFor1],1) DO
            IF __QUERYINTERFACE(groups[diFor1][diFor2], TEMP_ITF_CIRCUIT) THEN
				TEMP_ITF_CIRCUIT.set_release(en_static_define_state_off);
				TEMP_ITF_CIRCUIT.set_release_substate(en_static_define_sub_state_off);
				TEMP_ITF_CIRCUIT.set_release_next(en_release_next);

            ELSIF __QUERYINTERFACE(groups[diFor1][diFor2], TEMP_ITF_HYDRA) THEN
                (* Check if member is part of any other released circuit before turning off *)
                lock_if_released_in_other_circuit := FALSE;
                FOR diFor3 := LOWER_BOUND(groups,1) TO UPPER_BOUND(groups,1) DO
                    IF TEMP_ITF_HYDRA.MEMBER_OF(TO_USINT(diFor3)) AND groups_en_release[diFor3] = en_release THEN
                        lock_if_released_in_other_circuit := TRUE;
                    END_IF;
                END_FOR;
                IF NOT lock_if_released_in_other_circuit THEN
					TEMP_ITF_HYDRA.set_release(en_static_define_state_off);
					TEMP_ITF_HYDRA.set_release_substate(en_static_define_sub_state_off);
					TEMP_ITF_HYDRA.set_release_next(en_release_next);
                END_IF;
            END_IF;
        END_FOR;
    END_IF;
END_FOR;
END_ACTION

ACTION LOCKDOWN:
(* Get Status LockDown Engine*)
uiCountEngineLockDownOld := uiCountEngineLockDown;
uiCountEngineLockDown := 0;
FOR diFor1 := LOWER_BOUND(groups,1) TO UPPER_BOUND(groups,1) DO
	IF __QUERYINTERFACE(groups[diFor1][LOWER_BOUND(groups[diFor1],1)],TEMP_ITF_CIRCUIT) THEN
		uiCountEngineLockDown := uiCountEngineLockDown + TEMP_ITF_CIRCUIT.GET_ANZ_LOCKDOWN;
	END_IF;
END_FOR;
END_ACTION

ACTION AVAIABLE:
(* ------------------------------------------------------------- *)
(* Reset-Phase: Initialisierung der Gruppenstatusvariablen       *)
(* ------------------------------------------------------------- *)
FOR diFor1 := LOWER_BOUND(groups, 1) TO UPPER_BOUND(groups, 1) DO
	groups_en_available[diFor1]          := en_check;          // Setze Grundverfügbarkeit
	groups_en_available_substate[diFor1] := en_check_substate; // Setze Substate
END_FOR;


(* ------------------------------------------------------------- *)
(* Ermittlung des tatsächlichen Status jeder Gruppe              *)
(* ------------------------------------------------------------- *)
FOR diFor1 := LOWER_BOUND(groups, 1) TO UPPER_BOUND(groups, 1) DO
	// Durchlaufe alle Elemente innerhalb der Gruppe
	FOR diFor2 := LOWER_BOUND(groups[diFor1], 1) TO UPPER_BOUND(groups[diFor1], 1) DO
		
		// Überprüfe, ob Objekt gültig ist (Interface-Abfrage)
		IF __QUERYINTERFACE(groups[diFor1][diFor2], groups[diFor1][diFor2]) THEN
			
			// Nur relevante Objekte berücksichtigen
			IF NOT groups[diFor1][diFor2].IS_NOT_RELEVANT_TO_CHECK THEN
				
				// Wenn ein Element nicht den erwarteten Status hat → gesamte Gruppe auf "avaiable des abnormalen"
				IF groups[diFor1][diFor2].available <> en_check AND 
				   groups[diFor1][diFor2].available_substate = en_check_substate THEN
					
					groups_en_available[diFor1]          := groups[diFor1][diFor2].available;
					groups_en_available_substate[diFor1] := en_check_substate;
					
				END_IF;
			END_IF;
		// Prüfe ob Leader vorhanden
		ELSIF diFor2 = 0 THEN
			groups_en_available[diFor1]          := en_static_define_state_off;
			groups_en_available_substate[diFor1] := en_static_define_sub_state_off;	
		END_IF;
	END_FOR;
	
	// Versuche, aus der Gruppe die Anzahl verfügbarer Engines zu ermitteln
	IF __QUERYINTERFACE(groups[diFor1][LOWER_BOUND(groups[diFor1],1)], TEMP_ITF_CIRCUIT) THEN
		groups_engine_avaiable[diFor1] := TO_INT(TEMP_ITF_CIRCUIT.GET_ANZ_AVAIABLE);
	ELSE
		groups_engine_avaiable[diFor1] := 0; // 0 verfügbar
	END_IF;
END_FOR;


(* ------------------------------------------------------------- *)
(* Aggregation: Bestimme Gesamtstatus des Managers               *)
(* ------------------------------------------------------------- *)
en_available := en_static_define_lockdown; // Standardmäßig "ausfall"
FOR diFor1 := LOWER_BOUND(groups, 1) TO UPPER_BOUND(groups, 1) DO
	// Wenn mindestens eine Gruppe verfügbar ist, wird der Manager als "verfügbar" markiert
	IF groups_en_available[diFor1] = en_check AND groups_en_available_substate[diFor1] = en_check_substate THEN
		en_available          := en_check;
		en_available_substate := en_check_substate;
	END_IF;
END_FOR;


(* ------------------------------------------------------------- *)
(* Summierung: Gesamtanzahl verfügbarer Engines *)
(* ------------------------------------------------------------- *)
iAvaiable := 0;
FOR diFor1 := LOWER_BOUND(groups, 1) TO UPPER_BOUND(groups, 1) DO
	iAvaiable := iAvaiable + groups_engine_avaiable[diFor1];
END_FOR;
END_ACTION

METHOD ADD_CLIENT : BOOL
VAR_INPUT
	ITF_GROUP_BASE_IN	:	ITF_GROUPBASE;
END_VAR
VAR
	ITF_CIRCUIT_QUERRY	:	ITF_CIRCUIT;
	usiCircuitNr		:	USINT;
	ITF_HYDRA_QUERRY	:	ITF_HYDRA;
	xFailToAdd			:	BOOL;
	xExist				:	BOOL;
	xRegroup			:	BOOL;
	diForTemp1			:	DINT;
	diForTemp2			:	DINT;
	diForTemp3			:	DINT;
	diAddIn				:	DINT;
END_VAR
(* ADD CIRCUIT *)
IF __QUERYINTERFACE(ITF_GROUP_BASE_IN,ITF_CIRCUIT_QUERRY) THEN
	usiCircuitNr := ITF_CIRCUIT_QUERRY.CIRCUIT_NR;
	IF usiCircuitNr >= 1 AND usiCircuitNr <= GVL_CONSTANT.MAX_GROUPS THEN 
		IF groups[usiCircuitNr][0] = 0 THEN
			__QUERYINTERFACE(ITF_CIRCUIT_QUERRY,groups[usiCircuitNr][0]);
		ELSIF groups[usiCircuitNr][0] = ITF_GROUP_BASE_IN THEN
			ADD_CLIENT := TRUE;	
		ELSE
			ADD_CLIENT := FALSE;
		END_IF;
	END_IF;
(* ADD HYDRA *)
ELSIF __QUERYINTERFACE(ITF_GROUP_BASE_IN,ITF_HYDRA_QUERRY) THEN
	(* Check if is ADDED *)
	IF NOT ITF_HYDRA_QUERRY.IS_ADDED_TO_NESSESARY THEN
		FOR diForTemp1 := LOWER_BOUND(groups,1) TO UPPER_BOUND(groups,1) DO
			(* Reset Exist *)
			xExist := FALSE;
			(* Get Group Member *)
			IF ITF_HYDRA_QUERRY.MEMBER_OF(TO_USINT(diForTemp1)) THEN
				FOR diForTemp2 := LOWER_BOUND(groups[diForTemp1],1) TO UPPER_BOUND(groups[diForTemp1],1) DO
					IF groups[diForTemp1][diForTemp2] = ITF_GROUP_BASE_IN THEN
						xExist  := TRUE;
					END_IF;
				END_FOR;
				(* Add if not Exist *)
				IF NOT xExist THEN 
					IF aydiSyncG[diForTemp1] <> 0 THEN
						diAddIn  := __XADD(ADR(aydiSyncG[diForTemp1]),1);
						IF diAddIn >= 1 AND diAddIn <= UPPER_BOUND(groups[diForTemp1],1) THEN
							__QUERYINTERFACE(ITF_HYDRA_QUERRY,groups[diForTemp1][diAddIn]);
						ELSE
							xFailToAdd := TRUE;	
							ADD_CLIENT := FALSE;
						END_IF
					ELSE	
						xFailToAdd := TRUE;
						ADD_CLIENT := FALSE;
					END_IF;
				END_IF;
			ELSE
				FOR diForTemp2 := LOWER_BOUND(groups[diForTemp1],1) TO UPPER_BOUND(groups[diForTemp1],1) DO
					IF groups[diForTemp1][diForTemp2] = ITF_GROUP_BASE_IN THEN
						groups[diForTemp1][diForTemp2] := 0;
						FOR diForTemp3 := diForTemp2 TO UPPER_BOUND(groups[diForTemp1],1)-1 DO 
							groups[diForTemp1][diForTemp3] := groups[diForTemp1][diForTemp3+1];	
						END_FOR
						diAddIn  := __XADD(ADR(aydiSyncG[diForTemp1]),-1);
					END_IF;
				END_FOR;				
			END_IF
		END_FOR;
		ITF_HYDRA_QUERRY.IS_ADDED_TO_NESSESARY := NOT xFailToAdd;
	END_IF;	
ELSE
	ADD_CLIENT := FALSE;
END_IF;
END_METHOD

ACTION actParameter:
fbConfigFile();

scParameter.fbiTypeOfEngineManagement	(_usiParaNr := 1,	_WertInit := 0,		_MinInit := 0,	_MaxInit := 2,	itfConfigFb := fbConfigFile);
scParameter.fbtZuschaltSperrzeit		(_usiParaNr := 2,	_WertInit := T#5M,	_MinInit :=  ,	_MaxInit :=	 ,	itfConfigFb := fbConfigFile);
END_ACTION

END_FUNCTION_BLOCK

// 30 Program Organization Units/Manager/MANAGER_2
FUNCTION_BLOCK MANAGER_2 IMPLEMENTS ITF_MANAGER
VAR_INPUT
    en_check                                        : INT;   // Haupt-Check-State für die Engine-/Gruppenprüfung
    en_check_substate                               : INT;   // Substate des Check-Prozesses

    xRelease                                        : BOOL;  // BOOL-Trigger für eine Release-Anforderung
    iRelease                                        : INT;   // Integer-Releasewert oder Release-Kommando
    rRelease                                        : REAL;  // Realwert für Release-Parameter (z. B. Sollwert)

    en_release                                      : INT;   // Haupt-State des Release-Vorgangs
    en_release_substate                             : INT;   // Substate des Release-Vorgangs
    en_release_next                                 : INT;   // Nächster Release-State (State-Machine)

    scHzRelease                                     : CtaSysTypes.scHzParameter;  // Release-Parameter mit Hz-Information

    en_static_define_state_off                      : INT;   // Definierter State für OFF-Zustand
    en_static_define_sub_state_off                  : INT;   // Definierter Substate für OFF-Zustand
    en_static_define_lockdown                       : INT;   // State für Lockdown-Bedingungen
    en_static_define_substate_check_new_state       : INT;   // Substate zur Prüfung eines neuen State
    en_static_define_engine_release_from_substate   : INT;   // Substate, wenn Engine in Release-ON gehen soll
	en_static_define_engine_release_off_substate    : INT;   // Substate, wenn Engine in Release-OFF gehen soll
END_VAR

VAR_OUTPUT
    iAvaiable                                       : INT;   // Verfügbarkeitskennzahl der Engine/Gruppe
    en_available                                    : INT;   // Haupt-State der Verfügbarkeit
    en_available_substate                           : INT;   // Substate der Verfügbarkeit

    iAcknowledge                                    : INT;   // Integer-Wert zur Acknowledge-Verarbeitung
    rAcknowledge                                    : REAL;  // Realwert für Acknowledge-Parameter
    en_acknowledge                                  : INT;   // State für Acknowledge-Vorgang
    en_acknowledge_substate                         : INT;   // Substate des Acknowledge-Vorgangs

    en_demand                                       : INT;   // Haupt-State für Demand-/Anforderung
    en_demand_substate                              : INT;   // Substate für Demand-/Anforderung
    
    ITF_MANAGER                                     : ITF_MANAGER; // Manager-Interface für Gruppen-/Engine-Steuerung
END_VAR

VAR
    aydiSyncG                                       : ARRAY[1..GVL_CONSTANT.MAX_GROUPS] OF DINT := [GVL_CONSTANT.MAX_GROUPS(1)];
                                                        // Array zur Synchronisationsverwaltung der Gruppen

    groups                                          : ARRAY[1..GVL_CONSTANT.MAX_GROUPS] OF ARRAY[0..40] OF ITF_GROUPBASE;
                                                        // Struktur aller Gruppen und ihrer Members

    groups_en_available                             : ARRAY[1..GVL_CONSTANT.MAX_GROUPS] OF INT; // Verfügbarkeits-State je Gruppe
    groups_en_available_old                         : ARRAY[1..GVL_CONSTANT.MAX_GROUPS] OF INT; // Vorheriger Verfügbarkeits-State
    groups_en_available_substate                    : ARRAY[1..GVL_CONSTANT.MAX_GROUPS] OF INT; // Verfügbarkeits-Substate je Gruppe
    groups_en_available_substate_old                : ARRAY[1..GVL_CONSTANT.MAX_GROUPS] OF INT; // Alter Substate

    groups_engine_avaiable                          : ARRAY[1..GVL_CONSTANT.MAX_GROUPS] OF INT; // Engine-Verfügbarkeitsstate je Gruppe

    groups_en_acknowledge                           : ARRAY[1..GVL_CONSTANT.MAX_GROUPS] OF INT; // Acknowledge-State je Gruppe
    groups_en_acknowledge_old                       : ARRAY[1..GVL_CONSTANT.MAX_GROUPS] OF INT; // Alter Acknowledge-State
    groups_en_acknowledge_substate                  : ARRAY[1..GVL_CONSTANT.MAX_GROUPS] OF INT; // Acknowledge-Substate je Gruppe
    groups_en_acknowledge_substate_old              : ARRAY[1..GVL_CONSTANT.MAX_GROUPS] OF INT; // Alter Acknowledge-Substate

    groups_engine_acknowledge                       : ARRAY[1..GVL_CONSTANT.MAX_GROUPS] OF INT; // Engine-Acknowledge-State je Gruppe

    groups_en_release                               : ARRAY[1..GVL_CONSTANT.MAX_GROUPS] OF INT; // Release-State je Gruppe

    AY_GROUPS_AyPosMaxCT                            : ARRAY[1..GVL_CONSTANT.MAX_GROUPS] OF DINT; // Max-CT-Werte der Gruppen
    AY_GROUPS_xReleaseCircuit                       : ARRAY[1..GVL_CONSTANT.MAX_GROUPS] OF BOOL; // Release-Freigabe je Circuit

    TEMP_ITF_GROUPBASE                              : ITF_GROUPBASE; // Temp-Objekt für Gruppenoperationen
    TEMP_ITF_CIRCUIT                                : ITF_CIRCUIT;    // Temp-Circuit-Objekt
    TEMP_ITF_HYDRA                                  : ITF_HYDRA;      // Temp-Hydra-Objekt
    TEMP_ITF_HYDRA_MAX_CT                           : ITF_HYDRA;      // Temp-Hydra Objekt für max CT-Ermittlung

    diTempMemberCount                                : DINT;  // Temporäre Anzahl an Gruppenmitgliedern
    diFor1                                           : DINT;  // Schleifenzähler 1
    diFor2                                           : DINT;  // Schleifenzähler 2
    diFor3                                           : DINT;  // Schleifenzähler 3
    diNextCircuitToRun                               : DINT;  // Nächster Circuit, der gestartet werden soll
    diNextEngineToRun                                : DINT;  // Nächste Engine, die starten soll
    diNextCircuitToOff                               : DINT;  // Nächster Circuit zum Ausschalten
    diNextEngineToOff                                : DINT;  // Nächste Engine zum Ausschalten

    xTrigOn                                          : BOOL;  // Trigger für Start-/ON-Übergang
    xTrigOff                                         : BOOL;  // Trigger für Stop-/OFF-Übergang
    iTrigOffCount                                    : INT;   // Zähler für OFF-Triggerpflege
    iTrigOffMax                                      : INT;   // Maximal zulässige OFF-Triggerzeit

    enCheckOld                                       : INT;   // Alter Check-State
    enReleaseOld                                     : INT;   // Alter Release-State

    uiCountGroupLockDown                             : UINT;  // Anzahl Gruppen im Lockdown
    uiCountEngineLockDown                            : UINT;  // Anzahl Engines im Lockdown
    uiCountEngineAcknowledge                         : UINT;  // Anzahl Engines, die Acknowledge benötigen
    uiCountGroupLockDownOld                          : UINT;  // Vorherige Lockdown-Gruppenzahl
    uiCountEngineAcknowledgeOld                      : UINT;  // Vorherige Anzahl Acknowledge-Engines
    uiCountEngineLockDownOld                         : UINT;  // Vorherige Lockdown-Enginezahl

    iReleaseOld                                      : INT;   // Alter Releasewert
    iAcknowledgeOld                                  : INT;   // Alter Acknowledgewert

    xReleaseStopp                                    : BOOL;  // Stopp-Bedingung für Release
    TP_ReleaseLock                                   : Standard.TP;   // Timerbaustein für Release-Lock
    xResettReleaseLock_VIS                           : BOOL;  // Reset über VIS zum ReleaseLock

    lock_if_released_in_other_circuit                : BOOL;  // Lock, wenn Release in anderem Circuit aktiv ist

    // Parameter
    fbConfigFile                                     : CtaSysConfig.fbConfigFile; // Konfigurationsdatei-Handler
    scParameter                                      : scParameter;               // Parametrierobjekt
END_VAR

actParameter();

(* ITF *)
ITF_MANAGER := THIS^;

(* CHECK *)
CHECK();

(* AVAIABLE *)
AVAIABLE(); 

(* LOCKDOWN *)
LOCKDOWN();

(* ACKNOWLEDGE *)
ACKNOWLEDGE();

(* MANAGEMENT *)
MANAGEMENT();

(* RELEASE *)
RELEASE();

(* CHECK CHANGE *)
CHECK_RELEASE_CHANGE();

(* UPDATE *)
UPDATE_AT_THE_END();

ACTION CHECK:
(* Set Check State *)
FOR diFor1 := LOWER_BOUND(groups,1) TO UPPER_BOUND(groups,1) DO
	FOR diFor2 := LOWER_BOUND(groups[diFor1],1) TO UPPER_BOUND(groups[diFor1],1) DO
		IF __QUERYINTERFACE(groups[diFor1][diFor2],TEMP_ITF_GROUPBASE) THEN
			TEMP_ITF_GROUPBASE.set_check			(en_check);
			TEMP_ITF_GROUPBASE.set_check_substate	(en_check_substate);
		END_IF;
	END_FOR;
END_FOR;
END_ACTION

METHOD GET_NEXT_ENGINE_TO_RUN 
VAR_INPUT
	enTYPE_OF_ENGINE_MANAGEMENT	:	TYPE_OF_ENGINE_MANAGEMENT;
END_VAR
VAR_OUTPUT
	diNextCircuitToRunOut  		: DINT;
	diNextEngineToRunOut		: DINT;	
END_VAR
VAR 
	_diNextCircuitToRun  		: DINT;
	_diEngineLowestRunTime		: DINT;
	_xAvaiable					: BOOL;
	_xRelease					: BOOL;
	_rRelease					: REAL;
	_xAcknowledge				: BOOL;
	_rAcknowledge				: REAL;
	_xLockDown					: BOOL;
	_udiRunTime		    		: UDINT;
	_udiRunTimeTillOn   		: UDINT;
	_udiMinRunTime				: UDINT;
	_uiLowestWorkloadCircuit	: UINT;
END_VAR
(* Set Min Run Time To Max *)
_udiMinRunTime := 16#FFFFFFFF;
(* Set Lowest Workload Circuit to MAX *)
_uiLowestWorkloadCircuit := 16#FFFF;
(* Set Circuit to 0 *)
_diNextCircuitToRun := 0;
diNextCircuitToRunOut := 0;
(* Set Engine to 0  *)
_diEngineLowestRunTime := 0;
diNextEngineToRunOut := 0;

IF enTYPE_OF_ENGINE_MANAGEMENT = TYPE_OF_ENGINE_MANAGEMENT.RUN_1BY1 THEN
	FOR diFor1 := UPPER_BOUND(groups,1) TO LOWER_BOUND(groups,1) BY -1 DO 
		(* If No Error avaiable to release*)
		IF groups_en_available[diFor1] = en_release  OR groups_en_acknowledge[diFor1] = en_release THEN		
			IF __QUERYINTERFACE(groups[diFor1][LOWER_BOUND(groups[diFor1],1)],TEMP_ITF_CIRCUIT) THEN
				IF TEMP_ITF_CIRCUIT.GET_ANZ_RELEASE > 0 AND TEMP_ITF_CIRCUIT.GET_ANZ_AVAIABLE > 0 THEN
					(* iterate Engine and Check if Avaiable and get the Minits *)
					FOR diFor2 := TEMP_ITF_CIRCUIT.UPPERBOUND TO TEMP_ITF_CIRCUIT.LOWERBOUND BY -1 DO
						TEMP_ITF_CIRCUIT.GET_ENGINE_STATE(	usiNr 			:= TO_USINT(diFor2),
															xAvaiable 		=> _xAvaiable,
															xRelease		=> _xRelease,
															rRelease		=> _rRelease,
															xAcknowledge 	=> _xAcknowledge,
															rAcknowledge 	=> _rAcknowledge,
															xLockDown 		=> _xLockDown,
															udiRunTime 		=> _udiRunTime,
															udiRunTimeTillOn=> _udiRunTimeTillOn);
						(* Get time if Avaiable *)
						IF _xAvaiable AND NOT _xRelease AND NOT _xLockDown THEN
							IF _udiRunTime <= _udiMinRunTime THEN
								_udiMinRunTime 			:= _udiRunTime;
								_diNextCircuitToRun 	:= diFor1;
								_diEngineLowestRunTime  := diFor2;
							END_IF;			
						END_IF;						
					END_FOR;
				END_IF;
			END_IF;
		END_IF;
	END_FOR;
	(* Get new Ccuit if not possible to add ad running circuti *)
	IF _diNextCircuitToRun = 0 AND _diEngineLowestRunTime = 0  THEN
		FOR diFor1 := UPPER_BOUND(groups,1) TO LOWER_BOUND(groups,1) BY -1 DO
			(* If No Error avaiable to release*)
			IF groups_en_available[diFor1] = en_release  OR groups_en_acknowledge[diFor1] = en_release THEN	
				IF __QUERYINTERFACE(groups[diFor1][LOWER_BOUND(groups[diFor1],1)],TEMP_ITF_CIRCUIT) THEN
					IF TEMP_ITF_CIRCUIT.GET_ANZ_AVAIABLE > 0 THEN
						(* iterate Engine and Check if Avaiable and get the Minits *)
						FOR diFor2 := TEMP_ITF_CIRCUIT.UPPERBOUND TO TEMP_ITF_CIRCUIT.LOWERBOUND BY -1 DO
							TEMP_ITF_CIRCUIT.GET_ENGINE_STATE(	usiNr 			:= TO_USINT(diFor2),
																xAvaiable 		=> _xAvaiable,
																xRelease		=> _xRelease,
																rRelease		=> _rRelease,
																xAcknowledge 	=> _xAcknowledge,
																rAcknowledge 	=> _rAcknowledge,
																xLockDown 		=> _xLockDown,
																udiRunTime 		=> _udiRunTime,
																udiRunTimeTillOn=> _udiRunTimeTillOn);
							(* Get time if Avaiable *)
							IF _xAvaiable AND NOT _xRelease AND NOT _xLockDown THEN
								IF _udiRunTime <= _udiMinRunTime THEN
									_udiMinRunTime 			:= _udiRunTime;
									_diNextCircuitToRun 	:= diFor1;
									_diEngineLowestRunTime  := diFor2;
								END_IF;			
							END_IF;						
						END_FOR;
					END_IF;
				END_IF;
			END_IF;
		END_FOR;		
	END_IF
(* EQUAL *)
ELSIF enTYPE_OF_ENGINE_MANAGEMENT = TYPE_OF_ENGINE_MANAGEMENT.RUN_EQUAL THEN
	FOR diFor1 := UPPER_BOUND(groups,1) TO LOWER_BOUND(groups,1) BY -1 DO 
		(* If No Error avaiable to release*)
		IF groups_en_available[diFor1] = en_release  OR groups_en_acknowledge[diFor1] = en_release THEN	
			IF __QUERYINTERFACE(groups[diFor1][LOWER_BOUND(groups[diFor1],1)],TEMP_ITF_CIRCUIT) THEN
				IF TEMP_ITF_CIRCUIT.GET_ANZ_RELEASE <= _uiLowestWorkloadCircuit AND TEMP_ITF_CIRCUIT.GET_ANZ_AVAIABLE > 0 THEN
					_uiLowestWorkloadCircuit := TEMP_ITF_CIRCUIT.GET_ANZ_RELEASE; 
					(* iterate Engine and Check if Avaiable and get the Minits *)
					FOR diFor2 := TEMP_ITF_CIRCUIT.UPPERBOUND TO TEMP_ITF_CIRCUIT.LOWERBOUND BY -1 DO
						TEMP_ITF_CIRCUIT.GET_ENGINE_STATE(	usiNr 			:= TO_USINT(diFor2),
															xAvaiable 		=> _xAvaiable,
															xRelease		=> _xRelease,
															rRelease		=> _rRelease,
															xAcknowledge 	=> _xAcknowledge,
															rAcknowledge 	=> _rAcknowledge,
															xLockDown 		=> _xLockDown,
															udiRunTime 		=> _udiRunTime,
															udiRunTimeTillOn=> _udiRunTimeTillOn);
						(* Get time if Avaiable *)
						IF _xAvaiable AND NOT _xRelease AND NOT _xLockDown THEN
							IF _udiRunTime <= _udiMinRunTime THEN
								_udiMinRunTime 			:= _udiRunTime;
								_diNextCircuitToRun 	:= diFor1;
								_diEngineLowestRunTime  := diFor2;
							END_IF;			
						END_IF;						
					END_FOR;
				END_IF;
			END_IF;
		END_IF;
	END_FOR;
END_IF;
diNextCircuitToRunOut 	:= _diNextCircuitToRun;
diNextEngineToRunOut	:= _diEngineLowestRunTime;
END_METHOD

METHOD GET_NEXT_ENGINE_TO_OFF 
VAR_INPUT
	enTYPE_OF_ENGINE_MANAGEMENT	:	TYPE_OF_ENGINE_MANAGEMENT;
END_VAR
VAR_OUTPUT
	diNextCircuitToOffOut  		: DINT;
	diNextEngineToOffOut		: DINT;	
END_VAR
VAR 
	_diNextCircuitToOff  		: DINT;
	_diEngineHighestRunTime		: DINT;
	_xAvaiable					: BOOL;
	_xRelease					: BOOL;
	_rRelease					: REAL;
	_xAcknowledge				: BOOL;
	_rAcknowledge				: REAL;
	_xLockDown					: BOOL;
	_udiRunTime		    		: UDINT;
	_udiRunTimeTillOn   		: UDINT;
	_udiMaxRunTimeTillOn		: UDINT;
	_uiHighestWorkloadCircuit	: UINT;
	_uiLowestWorkloadCircuit	: UINT;
END_VAR
(* Set Highest Workload Circuit to Min *)
_uiHighestWorkloadCircuit := 16#0000;
(* Set Lowest Workload Circuit to MAX *)
_uiLowestWorkloadCircuit := 16#FFFF;
(* Set Max Run Time To Min *)
_udiMaxRunTimeTillOn := 16#0000;
(* Set Circuit to 0 *)
_diNextCircuitToOff := 0;
diNextCircuitToOffOut := 0;
(* Set Engine to 0  *)
_diEngineHighestRunTime := 0;
diNextEngineToOffOut := 0;
(* 1By1 *)
IF enTYPE_OF_ENGINE_MANAGEMENT = TYPE_OF_ENGINE_MANAGEMENT.RUN_1BY1 THEN
	FOR diFor1 := UPPER_BOUND(groups,1) TO LOWER_BOUND(groups,1) BY -1 DO 
		(* If No Error avaiable to release*)
		IF groups_en_available[diFor1] = en_release  OR groups_en_acknowledge[diFor1] = en_release THEN	
			IF __QUERYINTERFACE(groups[diFor1][LOWER_BOUND(groups[diFor1],1)],TEMP_ITF_CIRCUIT) THEN
				IF TEMP_ITF_CIRCUIT.GET_ANZ_RELEASE > 0 THEN
					IF TEMP_ITF_CIRCUIT.GET_ANZ_RELEASE <= _uiLowestWorkloadCircuit THEN
						IF TEMP_ITF_CIRCUIT.GET_ANZ_RELEASE < _uiLowestWorkloadCircuit THEN
							_uiLowestWorkloadCircuit := TEMP_ITF_CIRCUIT.GET_ANZ_RELEASE; 
							(* Set Max Run Time To Min *)
							_udiMaxRunTimeTillOn := 16#0000;
						END_IF;

						(* iterate Engine and Check if Avaiable and get the Minits *)
						FOR diFor2 := TEMP_ITF_CIRCUIT.UPPERBOUND TO TEMP_ITF_CIRCUIT.LOWERBOUND BY -1 DO
							TEMP_ITF_CIRCUIT.GET_ENGINE_STATE(	usiNr 			:= TO_USINT(diFor2),
																xAvaiable 		=> _xAvaiable,
																xRelease		=> _xRelease,
																rRelease		=> _rRelease,
																xAcknowledge 	=> _xAcknowledge,
																rAcknowledge 	=> _rAcknowledge,
																xLockDown 		=> _xLockDown,
																udiRunTime 		=> _udiRunTime,
																udiRunTimeTillOn=> _udiRunTimeTillOn);
							(* Get time if Running *)
							IF _xRelease THEN
								IF _udiRunTimeTillOn >= _udiMaxRunTimeTillOn THEN
									_udiMaxRunTimeTillOn 	:= _udiRunTimeTillOn;
									_diNextCircuitToOff 	:= diFor1;
									_diEngineHighestRunTime := diFor2;
								END_IF;			
							END_IF;						
						END_FOR;
					END_IF;
				END_IF;
			END_IF;
		END_IF;
	END_FOR;
(* EQUAL *)
ELSIF enTYPE_OF_ENGINE_MANAGEMENT = TYPE_OF_ENGINE_MANAGEMENT.RUN_EQUAL THEN
	FOR diFor1 := UPPER_BOUND(groups,1) TO LOWER_BOUND(groups,1) BY -1 DO 
		(* If No Error avaiable to release*)
		IF groups_en_available[diFor1] = en_release OR groups_en_acknowledge[diFor1] = en_release THEN	
			IF __QUERYINTERFACE(groups[diFor1][LOWER_BOUND(groups[diFor1],1)],TEMP_ITF_CIRCUIT) THEN
				IF TEMP_ITF_CIRCUIT.GET_ANZ_RELEASE >= _uiHighestWorkloadCircuit THEN
					IF TEMP_ITF_CIRCUIT.GET_ANZ_RELEASE > _uiHighestWorkloadCircuit THEN
						_uiHighestWorkloadCircuit := TEMP_ITF_CIRCUIT.GET_ANZ_RELEASE; 
						(* Set Max Run Time To Min *)
						_udiMaxRunTimeTillOn := 16#0000;				
					END_IF;
					(* iterate Engine and Check if Avaiable and get the time *)
					FOR diFor2 := TEMP_ITF_CIRCUIT.UPPERBOUND TO TEMP_ITF_CIRCUIT.LOWERBOUND BY -1 DO
						TEMP_ITF_CIRCUIT.GET_ENGINE_STATE(	usiNr 			:= TO_USINT(diFor2),
															xAvaiable 		=> _xAvaiable,
															xRelease		=> _xRelease,
															rRelease		=> _rRelease,
															xAcknowledge 	=> _xAcknowledge,
															rAcknowledge 	=> _rAcknowledge,
															xLockDown 		=> _xLockDown,
															udiRunTime 		=> _udiRunTime,
															udiRunTimeTillOn=> _udiRunTimeTillOn);
						(* Get time if Running *)
						IF _xRelease THEN
							IF _udiRunTimeTillOn >= _udiMaxRunTimeTillOn THEN
								_udiMaxRunTimeTillOn 	:= _udiRunTimeTillOn;
								_diNextCircuitToOff 	:= diFor1;
								_diEngineHighestRunTime := diFor2;
							END_IF;			
						END_IF;						
					END_FOR;
				END_IF;
			END_IF;
		END_IF;
	END_FOR;
END_IF;
diNextCircuitToOffOut 	:= _diNextCircuitToOff;
diNextEngineToOffOut	:= _diEngineHighestRunTime;
END_METHOD

ACTION MANAGEMENT:
(* ------------------------------------------------------------- *)
(* Engine Trigger Logic: TRIG ON / TRIG OFF and Release Handling   *)
(* ------------------------------------------------------------- *)

(* Wait until no TRIG ON is active, then determine next engine to run *)
IF NOT xTrigOn THEN
    GET_NEXT_ENGINE_TO_RUN(
        enTYPE_OF_ENGINE_MANAGEMENT := scParameter.fbiTypeOfEngineManagement.proValue,
        diNextCircuitToRunOut => diNextCircuitToRun,
        diNextEngineToRunOut  => diNextEngineToRun
    );
END_IF;

(* Wait until no TRIG OFF is active, then determine next engine to stop *)
IF NOT xTrigOff THEN
    GET_NEXT_ENGINE_TO_OFF(
        enTYPE_OF_ENGINE_MANAGEMENT := scParameter.fbiTypeOfEngineManagement.proValue,
        diNextCircuitToOffOut => diNextCircuitToOff,
        diNextEngineToOffOut  => diNextEngineToOff
    );
END_IF;

(* Check if engine is available and TRIG ON conditions are met *)
IF diNextCircuitToRun > 0 AND diNextEngineToRun > 0 THEN
    IF xRelease AND iRelease > 0 AND NOT xReleaseStopp THEN

        (* Handle group lockdown events *)
        IF uiCountGroupLockDown > uiCountGroupLockDownOld AND en_acknowledge <> en_static_define_lockdown THEN
            xTrigOn := TRUE;
            TP_ReleaseLock(IN := FALSE);

        (* Handle engine lockdown events *)
        ELSIF uiCountEngineLockDown > uiCountEngineLockDownOld AND en_acknowledge <> en_static_define_lockdown THEN
            xTrigOn := TRUE;
            TP_ReleaseLock(IN := FALSE);

        (* Handle engine turning off unexpectedly *)
        ELSIF uiCountEngineAcknowledge < uiCountEngineAcknowledgeOld AND iRelease > TO_INT(uiCountEngineAcknowledge) AND en_acknowledge <> en_static_define_lockdown THEN
            xTrigOn := TRUE;
            TP_ReleaseLock(IN := FALSE);

        (* Normal case: Add engine if release request exceeds acknowledge and no lock active *)
        ELSIF iRelease > iAcknowledge AND NOT TP_ReleaseLock.Q AND NOT xTrigOn THEN
            TP_ReleaseLock(IN := FALSE); (* Reset pulse before trigger *)
            xTrigOn := TRUE;
        END_IF;

    ELSE
        xTrigOn := FALSE; (* Release not active → no TRIG ON *)
    END_IF;
END_IF;

(* Manage normal release lock timer with minimum of 60s *)
IF NOT xResettReleaseLock_VIS AND xRelease THEN
    IF scParameter.fbtZuschaltSperrzeit.proValue > T#60S THEN
        TP_ReleaseLock(PT := scParameter.fbtZuschaltSperrzeit.proValue);
    ELSE
        TP_ReleaseLock(PT := T#60S);
    END_IF;
ELSE
    TP_ReleaseLock(IN := FALSE, PT := T#0MS);
    xResettReleaseLock_VIS := FALSE;
END_IF;

(* Check if engine is available and TRIG OFF conditions are met *)
IF diNextCircuitToOff > 0 AND diNextEngineToOff > 0 THEN
    IF xRelease THEN

        (* Reset case: Release equals acknowledge → reset counters *)
        IF iRelease = iAcknowledge THEN
            iTrigOffMax := 0;
            iTrigOffCount := 0;
            IF xTrigOn THEN (* Prevent endless engine running *)
                xTrigOn := FALSE;
                xTrigOff := TRUE;
                diNextCircuitToOff := diNextCircuitToRun;
                diNextEngineToOff  := diNextEngineToRun;
            END_IF

        (* Normal reduction: Release < acknowledge → trigger engine off *)
        ELSIF iRelease < iAcknowledge THEN
            IF iRelease < iReleaseOld OR iAcknowledge > iAcknowledgeOld THEN
                iTrigOffMax := MIN(iAcknowledge, iTrigOffMax + iReleaseOld - iRelease);
            END_IF
            IF iTrigOffCount < iTrigOffMax THEN
                iTrigOffCount := iTrigOffCount + 1;
                xTrigOff := TRUE;
            END_IF;
        END_IF;

    ELSE
        xTrigOff := FALSE; (* Release inactive → no TRIG OFF *)
    END_IF;
END_IF;

(* Set Release array and trigger engines accordingly *)
FOR diFor1 := LOWER_BOUND(groups,1) TO UPPER_BOUND(groups,1) DO
    IF __QUERYINTERFACE(groups[diFor1][LOWER_BOUND(groups[diFor1],1)], TEMP_ITF_CIRCUIT) THEN
        IF groups_en_acknowledge[diFor1] <> en_static_define_lockdown THEN
            IF TEMP_ITF_CIRCUIT.IS_RELEVANT_TO_RELEASE THEN

                (* Stop engine if it is next to be turned off *)
                IF diFor1 = diNextCircuitToOff AND xTrigOff THEN
                    TEMP_ITF_CIRCUIT.RELEASE_ENGINE(TO_USINT(diNextEngineToOff), FALSE);
                    xTrigOff := FALSE;
                    xTrigOn := FALSE;
                END_IF;

                (* Release engine if it is next to run and TRIG ON is active *)
                IF (groups_en_available[diFor1] = en_release OR groups_en_available[diFor1] = en_release_next OR groups_en_acknowledge[diFor1] = en_release) AND diFor1 = diNextCircuitToRun AND xTrigOn AND iRelease > 0 THEN
                    groups_en_release[diFor1] := en_release;
                    IF groups_en_acknowledge_substate[diFor1] >= en_static_define_engine_release_from_substate AND groups_en_acknowledge_substate[diFor1] <= en_static_define_engine_release_off_substate THEN
                        IF TEMP_ITF_CIRCUIT.IS_RELEVANT_TO_RELEASE AND AY_GROUPS_xReleaseCircuit[diFor1] THEN
							TEMP_ITF_CIRCUIT.RELEASE_ENGINE(TO_USINT(diNextEngineToRun), TRUE);
							xTrigOn := FALSE;
                        	TP_ReleaseLock(IN := TRUE);
						END_IF;
                    ELSE
                        TEMP_ITF_CIRCUIT.ALL_OFF();
                    END_IF;
                ELSIF groups_en_acknowledge[diFor1] = en_static_define_lockdown OR TEMP_ITF_CIRCUIT.GET_ANZ_RELEASE = 0 OR iRelease = 0 OR groups_en_acknowledge_substate[diFor1] < en_static_define_engine_release_from_substate OR groups_en_acknowledge_substate[diFor1] > en_static_define_engine_release_off_substate THEN
                    TEMP_ITF_CIRCUIT.ALL_OFF();
                    groups_en_release[diFor1] := en_static_define_state_off;
                END_IF;

            ELSE
                TEMP_ITF_CIRCUIT.ALL_OFF();
                groups_en_release[diFor1] := en_release;
            END_IF;
        ELSE
            TEMP_ITF_CIRCUIT.ALL_OFF();
            groups_en_release[diFor1] := en_static_define_state_off;
        END_IF;
    ELSE
        groups_en_release[diFor1] := en_static_define_state_off;
    END_IF;
END_FOR;

(* Apply HZ scale to relevant circuits *)
FOR diFor1 := LOWER_BOUND(groups,1) TO UPPER_BOUND(groups,1) DO
    IF __QUERYINTERFACE(groups[diFor1][LOWER_BOUND(groups[diFor1],1)], TEMP_ITF_CIRCUIT) THEN
        IF TEMP_ITF_CIRCUIT.IS_RELEVANT_TO_RELEASE THEN
            TEMP_ITF_CIRCUIT.SET_HZ_SCALE(scHzRelease);
        END_IF;
    END_IF;
END_FOR;

(* Set cyclic speed proportionally if acknowledge has not changed *)
IF iAcknowledge = iAcknowledgeOld THEN
    FOR diFor1 := LOWER_BOUND(groups,1) TO UPPER_BOUND(groups,1) DO
        IF __QUERYINTERFACE(groups[diFor1][LOWER_BOUND(groups[diFor1],1)], TEMP_ITF_CIRCUIT) THEN
            IF TEMP_ITF_CIRCUIT.IS_RELEVANT_TO_RELEASE THEN
                FOR diFor2 := TEMP_ITF_CIRCUIT.LOWERBOUND TO TEMP_ITF_CIRCUIT.UPPERBOUND DO
                    TEMP_ITF_CIRCUIT.prorRelease := rRelease;
                END_FOR;
            END_IF;
        END_IF;
    END_FOR;
END_IF;
END_ACTION

ACTION CHECK_RELEASE_CHANGE:
(* Not Avaiable if Changed *)
IF en_check <> enCheckOld THEN
	en_available := en_static_define_state_off;
END_IF;
END_ACTION

ACTION UPDATE_AT_THE_END:
iAcknowledgeOld := iAcknowledge;
enReleaseOld 	:= en_release;
enCheckOld	 	:= en_check;
iReleaseOld		:= iRelease;
END_ACTION

ACTION ACKNOWLEDGE:
(* ------------------------------------------------------------- *)
(* Reset Phase: Initialize group acknowledge status variables      *)
(* ------------------------------------------------------------- *)
FOR diFor1 := LOWER_BOUND(groups,1) TO UPPER_BOUND(groups,1) DO
    IF __QUERYINTERFACE(groups[diFor1][0], TEMP_ITF_CIRCUIT) THEN
        (* Set initial acknowledge state to release for circuits *)
        groups_en_acknowledge[diFor1] := en_release;
        groups_en_acknowledge_substate[diFor1] := en_release_substate;
    ELSE
        (* Set initial acknowledge state to off if no circuit *)
        groups_en_acknowledge[diFor1] := en_static_define_state_off;
        groups_en_acknowledge_substate[diFor1] := en_static_define_sub_state_off;
    END_IF;
END_FOR;

(* ------------------------------------------------------------- *)
(* Determine actual acknowledge status of each group               *)
(* ------------------------------------------------------------- *)
FOR diFor1 := LOWER_BOUND(groups,1) TO UPPER_BOUND(groups,1) DO
    (* Iterate over all members of the group *)
    FOR diFor2 := LOWER_BOUND(groups[diFor1],1) TO UPPER_BOUND(groups[diFor1],1) DO
        IF __QUERYINTERFACE(groups[diFor1][diFor2], groups[diFor1][diFor2]) THEN
            (* Only consider relevant objects for release and acknowledge *)
            IF NOT groups[diFor1][diFor2].IS_NOT_RELEVANT_TO_RELEASE AND NOT groups[diFor1][diFor2].IS_NOT_RELEVANT_TO_ACKNOWLEDGE THEN
                (* Update group acknowledge status based on member *)
                IF groups[diFor1][diFor2].acknowledge <> en_release THEN
                    IF groups[diFor1][diFor2].acknowledge = en_static_define_lockdown THEN
                        (* If this group was about to run, cancel TRIG ON *)
                        IF diNextCircuitToRun = diFor1 AND xTrigOn THEN
                            xTrigOn := FALSE;
                        END_IF;
                        groups_en_acknowledge[diFor1] := en_static_define_lockdown; (* Lockdown for group *)
                    ELSE
						IF groups_en_acknowledge[diFor1] <> en_static_define_lockdown THEN
                        	groups_en_acknowledge[diFor1] := groups[diFor1][diFor2].acknowledge;
						END_IF;
                    END_IF;
                END_IF;

                (* Update substate if it differs from release substate *)
                IF groups[diFor1][diFor2].acknowledge_substate <> en_release_substate THEN
                    groups_en_acknowledge_substate[diFor1] := groups[diFor1][diFor2].acknowledge_substate;
                END_IF;
            END_IF;
        END_IF;
    END_FOR;

    (* Count acknowledged engines per group if circuit interface is valid *)
    IF __QUERYINTERFACE(groups[diFor1][LOWER_BOUND(groups[diFor1],1)], TEMP_ITF_CIRCUIT) THEN
        groups_engine_acknowledge[diFor1] := TO_INT(TEMP_ITF_CIRCUIT.GET_ANZ_ACKNOWLEDGE);
    ELSE
        groups_engine_acknowledge[diFor1] := 0;
    END_IF;
END_FOR;

(* ------------------------------------------------------------- *)
(* Set acknowledge status for manager based on group status       *)
(* ------------------------------------------------------------- *)
en_acknowledge := 0;
FOR diFor1 := LOWER_BOUND(groups,1) TO UPPER_BOUND(groups,1) DO
    (* If any group is in lockdown, manager is in lockdown *)
    IF groups_en_acknowledge[diFor1] = en_static_define_lockdown THEN
        en_acknowledge := en_static_define_lockdown;
    END_IF;
END_FOR;

FOR diFor1 := LOWER_BOUND(groups,1) TO UPPER_BOUND(groups,1) DO
    (* If any group is in release and substate matches, update manager acknowledge *)
    IF groups_en_acknowledge[diFor1] = en_release OR ( groups_en_acknowledge[diFor1] <> en_static_define_lockdown AND groups_en_release[diFor1] = en_release ) THEN
		en_acknowledge := groups_en_acknowledge[diFor1];
        IF groups_en_acknowledge_substate[diFor1] = en_release_substate  THEN
            en_acknowledge_substate := en_release_substate;
        END_IF;		
    END_IF;
END_FOR;

(* Update engine acknowledge counters *)
iAcknowledge := 0;
uiCountEngineAcknowledgeOld := uiCountEngineAcknowledge;
FOR diFor1 := LOWER_BOUND(groups,1) TO UPPER_BOUND(groups,1) DO
    iAcknowledge := iAcknowledge + groups_engine_acknowledge[diFor1];
END_FOR;
uiCountEngineAcknowledge := TO_UINT(iAcknowledge);
END_ACTION

ACTION RELEASE:
(* Set Release for each group and its components *)
FOR diFor1 := LOWER_BOUND(groups,1) TO UPPER_BOUND(groups,1) DO

    (* Check if group is in release state and not in lockdown *)
    IF (groups_en_release[diFor1] = en_release OR groups_en_release[diFor1] = enReleaseOld) AND groups_en_acknowledge[diFor1] <> en_static_define_lockdown THEN
        (* Initially set group as ready for release *)
        AY_GROUPS_xReleaseCircuit[diFor1] := TRUE;

        (* Check each member in the group to verify readiness for release *)
        FOR diFor2 := LOWER_BOUND(groups[diFor1],1)+1 TO UPPER_BOUND(groups[diFor1],1) DO
            IF __QUERYINTERFACE(groups[diFor1][diFor2], TEMP_ITF_HYDRA) THEN
                IF NOT groups[diFor1][diFor2].IS_NOT_RELEVANT_TO_RELEASE AND NOT groups[diFor1][diFor2].IS_NOT_RELEVANT_TO_ACKNOWLEDGE THEN
                    IF groups[diFor1][diFor2].acknowledge <> en_release OR groups[diFor1][diFor2].acknowledge_substate <> en_static_define_engine_release_from_substate THEN
                        (* Member not ready, set group as not ready *)
                        AY_GROUPS_xReleaseCircuit[diFor1] := FALSE;
                    END_IF;
                END_IF;
            END_IF;
        END_FOR;

        (* Apply release settings to each relevant member of the group *)
        FOR diFor2 := LOWER_BOUND(groups[diFor1],1)+1 TO UPPER_BOUND(groups[diFor1],1) DO
            IF __QUERYINTERFACE(groups[diFor1][diFor2], groups[diFor1][diFor2]) THEN
                IF NOT groups[diFor1][diFor2].IS_NOT_RELEVANT_TO_RELEASE THEN
                    IF __QUERYINTERFACE(groups[diFor1][diFor2], TEMP_ITF_HYDRA) THEN
                        TEMP_ITF_HYDRA.set_release(en_release);
                        TEMP_ITF_HYDRA.set_release_substate(en_release_substate);
                        TEMP_ITF_HYDRA.set_release_next(en_release_next);
                    END_IF;
                ELSE
                    (* Member not relevant → set off *)
                    IF __QUERYINTERFACE(groups[diFor1][diFor2], TEMP_ITF_HYDRA) THEN
                        TEMP_ITF_HYDRA.set_release(en_static_define_state_off);
                        TEMP_ITF_HYDRA.set_release_substate(en_static_define_sub_state_off);
                        TEMP_ITF_HYDRA.set_release_next(en_release_next);
                    END_IF;
                END_IF;
            END_IF;
        END_FOR;

        (* Release settings for group leader *)
        IF groups[diFor1][LOWER_BOUND(groups[diFor1],1)] <> 0 THEN
            IF __QUERYINTERFACE(groups[diFor1][LOWER_BOUND(groups[diFor1],1)], TEMP_ITF_CIRCUIT) THEN
				TEMP_ITF_CIRCUIT.set_release(en_release);
				TEMP_ITF_CIRCUIT.set_release_substate(en_release_substate);
				TEMP_ITF_CIRCUIT.set_release_next(en_release_next);
			ELSE
				(* Leader not relevant → set off *)
				TEMP_ITF_CIRCUIT.set_release(en_release);
				TEMP_ITF_CIRCUIT.set_release_substate(en_release_substate);
				TEMP_ITF_CIRCUIT.set_release_next(en_release_next);
			END_IF;
        END_IF;

    ELSE
        (* Group not in release → mark as not ready *)
        AY_GROUPS_xReleaseCircuit[diFor1] := FALSE;

        (* Turn off all members of the group *)
        FOR diFor2 := LOWER_BOUND(groups[diFor1],1) TO UPPER_BOUND(groups[diFor1],1) DO
            IF __QUERYINTERFACE(groups[diFor1][diFor2], TEMP_ITF_CIRCUIT) THEN
				TEMP_ITF_CIRCUIT.set_release(en_static_define_state_off);
				TEMP_ITF_CIRCUIT.set_release_substate(en_static_define_sub_state_off);
				TEMP_ITF_CIRCUIT.set_release_next(en_release_next);

            ELSIF __QUERYINTERFACE(groups[diFor1][diFor2], TEMP_ITF_HYDRA) THEN
                (* Check if member is part of any other released circuit before turning off *)
                lock_if_released_in_other_circuit := FALSE;
                FOR diFor3 := LOWER_BOUND(groups,1) TO UPPER_BOUND(groups,1) DO
                    IF TEMP_ITF_HYDRA.MEMBER_OF(TO_USINT(diFor3)) AND groups_en_release[diFor3] = en_release THEN
                        lock_if_released_in_other_circuit := TRUE;
                    END_IF;
                END_FOR;
                IF NOT lock_if_released_in_other_circuit THEN
					TEMP_ITF_HYDRA.set_release(en_static_define_state_off);
					TEMP_ITF_HYDRA.set_release_substate(en_static_define_sub_state_off);
					TEMP_ITF_HYDRA.set_release_next(en_release_next);
                END_IF;
            END_IF;
        END_FOR;
    END_IF;
END_FOR;
END_ACTION

ACTION LOCKDOWN:
(* Get Status LockDown Engine*)
uiCountEngineLockDownOld := uiCountEngineLockDown;
uiCountEngineLockDown := 0;
FOR diFor1 := LOWER_BOUND(groups,1) TO UPPER_BOUND(groups,1) DO
	IF __QUERYINTERFACE(groups[diFor1][LOWER_BOUND(groups[diFor1],1)],TEMP_ITF_CIRCUIT) THEN
		uiCountEngineLockDown := uiCountEngineLockDown + TEMP_ITF_CIRCUIT.GET_ANZ_LOCKDOWN;
	END_IF;
END_FOR;
END_ACTION

ACTION AVAIABLE:
(* ------------------------------------------------------------- *)
(* Reset-Phase: Initialisierung der Gruppenstatusvariablen       *)
(* ------------------------------------------------------------- *)
FOR diFor1 := LOWER_BOUND(groups, 1) TO UPPER_BOUND(groups, 1) DO
	groups_en_available[diFor1]          := en_check;          // Setze Grundverfügbarkeit
	groups_en_available_substate[diFor1] := en_check_substate; // Setze Substate
END_FOR;


(* ------------------------------------------------------------- *)
(* Ermittlung des tatsächlichen Status jeder Gruppe              *)
(* ------------------------------------------------------------- *)
FOR diFor1 := LOWER_BOUND(groups, 1) TO UPPER_BOUND(groups, 1) DO
	// Durchlaufe alle Elemente innerhalb der Gruppe
	FOR diFor2 := LOWER_BOUND(groups[diFor1], 1) TO UPPER_BOUND(groups[diFor1], 1) DO
		
		// Überprüfe, ob Objekt gültig ist (Interface-Abfrage)
		IF __QUERYINTERFACE(groups[diFor1][diFor2], groups[diFor1][diFor2]) THEN
			
			// Nur relevante Objekte berücksichtigen
			IF NOT groups[diFor1][diFor2].IS_NOT_RELEVANT_TO_CHECK THEN
				
				// Wenn ein Element nicht den erwarteten Status hat → gesamte Gruppe auf "avaiable des abnormalen"
				IF groups[diFor1][diFor2].available <> en_check AND 
				   groups[diFor1][diFor2].available_substate = en_check_substate THEN
					
					groups_en_available[diFor1]          := groups[diFor1][diFor2].available;
					groups_en_available_substate[diFor1] := en_check_substate;
					
				END_IF;
			END_IF;
		// Prüfe ob Leader vorhanden
		ELSIF diFor2 = 0 THEN
			groups_en_available[diFor1]          := en_static_define_state_off;
			groups_en_available_substate[diFor1] := en_static_define_sub_state_off;	
		END_IF;
	END_FOR;
	
	// Versuche, aus der Gruppe die Anzahl verfügbarer Engines zu ermitteln
	IF __QUERYINTERFACE(groups[diFor1][LOWER_BOUND(groups[diFor1],1)], TEMP_ITF_CIRCUIT) THEN
		groups_engine_avaiable[diFor1] := TO_INT(TEMP_ITF_CIRCUIT.GET_ANZ_AVAIABLE);
	ELSE
		groups_engine_avaiable[diFor1] := 0; // 0 verfügbar
	END_IF;
END_FOR;


(* ------------------------------------------------------------- *)
(* Aggregation: Bestimme Gesamtstatus des Managers               *)
(* ------------------------------------------------------------- *)
en_available := en_static_define_lockdown; // Standardmäßig "ausfall"
FOR diFor1 := LOWER_BOUND(groups, 1) TO UPPER_BOUND(groups, 1) DO
	// Wenn mindestens eine Gruppe verfügbar ist, wird der Manager als "verfügbar" markiert
	IF groups_en_available[diFor1] = en_check AND groups_en_available_substate[diFor1] = en_check_substate THEN
		en_available          := en_check;
		en_available_substate := en_check_substate;
	END_IF;
END_FOR;


(* ------------------------------------------------------------- *)
(* Summierung: Gesamtanzahl verfügbarer Engines *)
(* ------------------------------------------------------------- *)
iAvaiable := 0;
FOR diFor1 := LOWER_BOUND(groups, 1) TO UPPER_BOUND(groups, 1) DO
	iAvaiable := iAvaiable + groups_engine_avaiable[diFor1];
END_FOR;
END_ACTION

METHOD ADD_CLIENT : BOOL
VAR_INPUT
	ITF_GROUP_BASE_IN	:	ITF_GROUPBASE;
END_VAR
VAR
	ITF_CIRCUIT_QUERRY	:	ITF_CIRCUIT;
	usiCircuitNr		:	USINT;
	ITF_HYDRA_QUERRY	:	ITF_HYDRA;
	xFailToAdd			:	BOOL;
	xExist				:	BOOL;
	xRegroup			:	BOOL;
	diForTemp1			:	DINT;
	diForTemp2			:	DINT;
	diForTemp3			:	DINT;
	diAddIn				:	DINT;
END_VAR
(* ADD CIRCUIT *)
IF __QUERYINTERFACE(ITF_GROUP_BASE_IN,ITF_CIRCUIT_QUERRY) THEN
	usiCircuitNr := ITF_CIRCUIT_QUERRY.CIRCUIT_NR;
	IF usiCircuitNr >= 1 AND usiCircuitNr <= GVL_CONSTANT.MAX_GROUPS THEN 
		IF groups[usiCircuitNr][0] = 0 THEN
			__QUERYINTERFACE(ITF_CIRCUIT_QUERRY,groups[usiCircuitNr][0]);
		ELSIF groups[usiCircuitNr][0] = ITF_GROUP_BASE_IN THEN
			ADD_CLIENT := TRUE;	
		ELSE
			ADD_CLIENT := FALSE;
		END_IF;
	END_IF;
(* ADD HYDRA *)
ELSIF __QUERYINTERFACE(ITF_GROUP_BASE_IN,ITF_HYDRA_QUERRY) THEN
	(* Check if is ADDED *)
	IF NOT ITF_HYDRA_QUERRY.IS_ADDED_TO_NESSESARY THEN
		FOR diForTemp1 := LOWER_BOUND(groups,1) TO UPPER_BOUND(groups,1) DO
			(* Reset Exist *)
			xExist := FALSE;
			(* Get Group Member *)
			IF ITF_HYDRA_QUERRY.MEMBER_OF(TO_USINT(diForTemp1)) THEN
				FOR diForTemp2 := LOWER_BOUND(groups[diForTemp1],1) TO UPPER_BOUND(groups[diForTemp1],1) DO
					IF groups[diForTemp1][diForTemp2] = ITF_GROUP_BASE_IN THEN
						xExist  := TRUE;
					END_IF;
				END_FOR;
				(* Add if not Exist *)
				IF NOT xExist THEN 
					IF aydiSyncG[diForTemp1] <> 0 THEN
						diAddIn  := __XADD(ADR(aydiSyncG[diForTemp1]),1);
						IF diAddIn >= 1 AND diAddIn <= UPPER_BOUND(groups[diForTemp1],1) THEN
							__QUERYINTERFACE(ITF_HYDRA_QUERRY,groups[diForTemp1][diAddIn]);
						ELSE
							xFailToAdd := TRUE;	
							ADD_CLIENT := FALSE;
						END_IF
					ELSE	
						xFailToAdd := TRUE;
						ADD_CLIENT := FALSE;
					END_IF;
				END_IF;
			ELSE
				FOR diForTemp2 := LOWER_BOUND(groups[diForTemp1],1) TO UPPER_BOUND(groups[diForTemp1],1) DO
					IF groups[diForTemp1][diForTemp2] = ITF_GROUP_BASE_IN THEN
						groups[diForTemp1][diForTemp2] := 0;
						FOR diForTemp3 := diForTemp2 TO UPPER_BOUND(groups[diForTemp1],1)-1 DO 
							groups[diForTemp1][diForTemp3] := groups[diForTemp1][diForTemp3+1];	
						END_FOR
						diAddIn  := __XADD(ADR(aydiSyncG[diForTemp1]),-1);
					END_IF;
				END_FOR;				
			END_IF
		END_FOR;
		ITF_HYDRA_QUERRY.IS_ADDED_TO_NESSESARY := NOT xFailToAdd;
	END_IF;	
ELSE
	ADD_CLIENT := FALSE;
END_IF;
END_METHOD

ACTION actParameter:
fbConfigFile();

scParameter.fbiTypeOfEngineManagement	(_usiParaNr := 1,	_WertInit := 0,		_MinInit := 0,	_MaxInit := 2,	itfConfigFb := fbConfigFile);
scParameter.fbtZuschaltSperrzeit		(_usiParaNr := 2,	_WertInit := T#5M,	_MinInit :=  ,	_MaxInit :=	 ,	itfConfigFb := fbConfigFile);
END_ACTION

END_FUNCTION_BLOCK

// 40 Visualizations/Dialog/DIA_MANAGERCONFIG
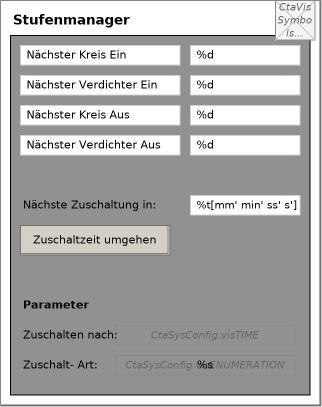
VISUALIZATION DIA_MANAGERCONFIG  // 322x407
VAR_IN_OUT
	{attribute 'VAR_IN_OUT_AS_POINTER'}
	MANAGER_DIA			:	MANAGER;
END_VAR
    RoundedRectangle (0,0 320x405)
    RoundedRectangle (10,35 300x360)
    Button (20,225 150x30), "Zuschaltzeit umgehen"
        toggle MANAGER_DIA.xResettReleaseLock_VIS
    Textfield (20,45 160x20), "Nächster Kreis Ein"
    Textfield (20,75 160x20), "Nächster Verdichter Ein"
    Textfield (20,135 160x20), "Nächster Verdichter Aus"
    Textfield (20,105 160x20), "Nächster Kreis Aus"
    Textfield (190,45 110x20), "%d", text variable: MANAGER_DIA.next_circuit_to_run_engine
    Textfield (190,75 110x20), "%d", text variable: MANAGER_DIA.next_engine_to_run
    Textfield (190,105 110x20), "%d", text variable: MANAGER_DIA.next_circuit_to_stopp_engine
    Textfield (190,135 110x20), "%d", text variable: MANAGER_DIA.next_engine_to_stopp
    Frame (115,325 180x20)
        shows CtaSysConfig.visTIME(visfbTIMEIn := MANAGER_DIA.scParameter.fbtZuschaltSperrzeit)
    Frame (115,355 180x20)
        shows CtaSysConfig.visENUMERATION(visfbENUIn := MANAGER_DIA.scParameter.fbiTypeOfEngineManagement)
    Label (20,325 150x20), "Zuschalten nach:"
    Label (20,355 150x20), "Zuschalt- Art:"
    Textfield (190,195 110x20), "%t[mm' min' ss' s']", text variable: (MANAGER_DIA.scParameter.fbtZuschaltSperrzeit.proValue - MANAGER_DIA.TP_ReleaseLock.ET)
    Textfield (20,195 160x20), "Nächste Zuschaltung in:"
    Textfield (20,295 160x20), "Parameter"
    Image (275,0 40x40), image: CtaVisSymbols.ImagePool.close_solo_black
        OnMouseClick:  Dialog=Current Dialog, Result=OK, NumpadKeypadSet=True
    Label (10,0 150x40), "Stufenmanager"
    Textfield (135,355 140x20), "%s", text list: 'TypeOfEngineManagement', text index: CtaSysConfig.fcGetEnumerationId(MANAGER_DIA.scParameter.fbiTypeOfEngineManagement)
END_VISUALIZATION

// 40 Visualizations/VIS_Manager_rEck
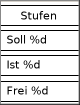
VISUALIZATION VIS_Manager_rEck  // 80x105
VAR_IN_OUT
	MANAGER_IN		:	MANAGER;
END_VAR
    Textfield (0,1 80x105)
    Textfield (0,6 78x20), "Stufen"
    Textfield (0,30 78x20), "Soll %d", text variable: MANAGER_IN.iRelease
    Textfield (0,55 78x20), "Ist %d", text variable: MANAGER_IN.iAcknowledged
    Textfield (0,81 78x20), "Frei %d", text variable: MANAGER_IN.iAvailableTemp
    Line (0,30) (79,30)
    Line (0,50) (79,50)
    Line (0,55) (79,55)
    Line (0,75) (79,75)
    Line (0,81) (79,81)
    Line (0,101) (79,101)
    Line (0,5) (79,5)
    Line (0,25) (79,25)
    Rectangle (0,0 80x105)
        OnMouseClick:  Dialog=DIA_MANAGERCONFIG, Parameters={MANAGER_DIA: MANAGER_IN}, Selected={0: }, OpenCentered=True
END_VISUALIZATION

// 40 Visualizations/VIS_Manager
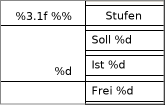
VISUALIZATION VIS_Manager  // 165x105
VAR_IN_OUT
	MANAGER_IN		:	MANAGER;
END_VAR
    Line (0,25) (157,25)
    Line (0,81) (158,81)
    Rectangle (15,65 60x13), "%d", text variable: MANAGER_IN.iRelease
    Rectangle (15,10 60x13), "%3.1f %%", text variable: MANAGER_IN.rRelease
    Frame (85,0 80x105)
        shows VIS_Manager_rEck(MANAGER_IN := MANAGER_IN)
END_VISUALIZATION

(* text list TypeOfEngineManagement (id | default | de | en | fr | it)
  0 | RUN 1BY1 |  |  |  | 
  1 | RUN EQUAL |  |  |  | 
   |  |  |  |  |  *)
